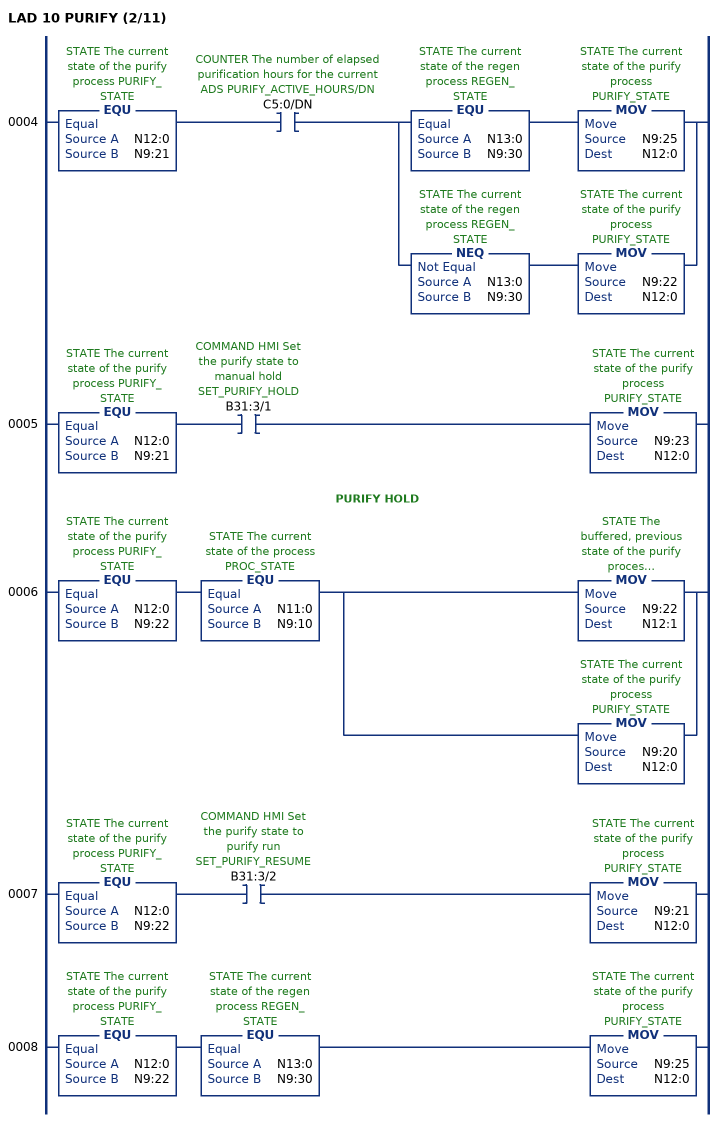
% Rung: 4 %
SOR EQU N12:0 N9:21 XIC C5:0/DN BST EQU N13:0 N9:30 MOV N9:25 N12:0 NXB NEQ N13:0 N9:30 MOV N9:22 N12:0 BND EOR
%   N12:0  PURIFY_STATE  "STATE The current state of the purify process" %
%   N9:21  PURIFY_RUN  "STATE Purify running" %
%   C5:0  PURIFY_ACTIVE_HOURS  "COUNTER The number of elapsed purification hours for the current ADS" %
%   N13:0  REGEN_STATE  "STATE The current state of the regen process" %
%   N9:30  REGEN_STANDBY  "STATE Regen Standby" %
%   N9:25  PURIFY_DONE %
%   N9:22  PURIFY_HOLD  "STATE Purify Hold" %
% Rung: 5 %
SOR EQU N12:0 N9:21 XIC B31:3/1 MOV N9:23 N12:0 EOR
%   N12:0  PURIFY_STATE  "STATE The current state of the purify process" %
%   N9:21  PURIFY_RUN  "STATE Purify running" %
%   B31:3/1  SET_PURIFY_HOLD  "COMMAND HMI Set the purify state to manual hold" %
%   N9:23  PURIFY_MANUAL_HOLD  "STATE Purify Manual Hold" %
% Rung: 6 %
% TITLE: PURIFY HOLD %
SOR EQU N12:0 N9:22 EQU N11:0 N9:10 BST MOV N9:22 N12:1 NXB MOV N9:20 N12:0 BND EOR
%   N12:0  PURIFY_STATE  "STATE The current state of the purify process" %
%   N9:22  PURIFY_HOLD  "STATE Purify Hold" %
%   N11:0  PROC_STATE  "STATE The current state of the process" %
%   N9:10  PROC_STANDBY  "STATE Process Standby" %
%   N12:1  PURIFY_STATE_BUFFER  "STATE The buffered, previous state of the purify process" %
%   N9:20  PURIFY_STANDBY  "STATE Purify Standby" %
% Rung: 7 %
SOR EQU N12:0 N9:22 XIC B31:3/2 MOV N9:21 N12:0 EOR
%   N12:0  PURIFY_STATE  "STATE The current state of the purify process" %
%   N9:22  PURIFY_HOLD  "STATE Purify Hold" %
%   B31:3/2  SET_PURIFY_RESUME  "COMMAND HMI Set the purify state to purify run" %
%   N9:21  PURIFY_RUN  "STATE Purify running" %
% Rung: 8 %
SOR EQU N12:0 N9:22 EQU N13:0 N9:30 MOV N9:25 N12:0 EOR
%   N12:0  PURIFY_STATE  "STATE The current state of the purify process" %
%   N9:22  PURIFY_HOLD  "STATE Purify Hold" %
%   N13:0  REGEN_STATE  "STATE The current state of the regen process" %
%   N9:30  REGEN_STANDBY  "STATE Regen Standby" %
%   N9:25  PURIFY_DONE %

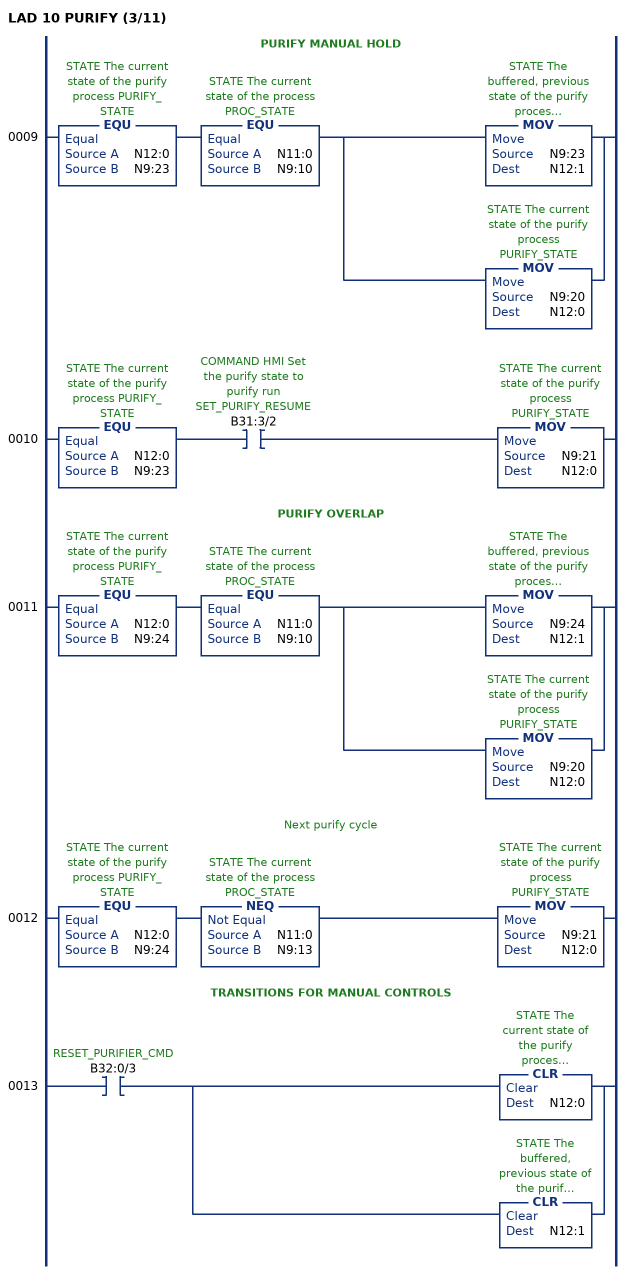
% Rung: 9 %
% TITLE: PURIFY MANUAL HOLD %
SOR EQU N12:0 N9:23 EQU N11:0 N9:10 BST MOV N9:23 N12:1 NXB MOV N9:20 N12:0 BND EOR
%   N12:0  PURIFY_STATE  "STATE The current state of the purify process" %
%   N9:23  PURIFY_MANUAL_HOLD  "STATE Purify Manual Hold" %
%   N11:0  PROC_STATE  "STATE The current state of the process" %
%   N9:10  PROC_STANDBY  "STATE Process Standby" %
%   N12:1  PURIFY_STATE_BUFFER  "STATE The buffered, previous state of the purify process" %
%   N9:20  PURIFY_STANDBY  "STATE Purify Standby" %
% Rung: 10 %
SOR EQU N12:0 N9:23 XIC B31:3/2 MOV N9:21 N12:0 EOR
%   N12:0  PURIFY_STATE  "STATE The current state of the purify process" %
%   N9:23  PURIFY_MANUAL_HOLD  "STATE Purify Manual Hold" %
%   B31:3/2  SET_PURIFY_RESUME  "COMMAND HMI Set the purify state to purify run" %
%   N9:21  PURIFY_RUN  "STATE Purify running" %
% Rung: 11 %
% TITLE: PURIFY OVERLAP %
SOR EQU N12:0 N9:24 EQU N11:0 N9:10 BST MOV N9:24 N12:1 NXB MOV N9:20 N12:0 BND EOR
%   N12:0  PURIFY_STATE  "STATE The current state of the purify process" %
%   N9:24  PURIFY_OVERLAP  "STATE Puriify Overlap" %
%   N11:0  PROC_STATE  "STATE The current state of the process" %
%   N9:10  PROC_STANDBY  "STATE Process Standby" %
%   N12:1  PURIFY_STATE_BUFFER  "STATE The buffered, previous state of the purify process" %
%   N9:20  PURIFY_STANDBY  "STATE Purify Standby" %
% Rung: 12 %
% Next purify cycle %
SOR EQU N12:0 N9:24 NEQ N11:0 N9:13 MOV N9:21 N12:0 EOR
%   N12:0  PURIFY_STATE  "STATE The current state of the purify process" %
%   N9:24  PURIFY_OVERLAP  "STATE Puriify Overlap" %
%   N11:0  PROC_STATE  "STATE The current state of the process" %
%   N9:13  PROC_OVERLAP  "STATE Process Purify Overlap" %
%   N9:21  PURIFY_RUN  "STATE Purify running" %
% Rung: 13 %
% TITLE: TRANSITIONS FOR MANUAL CONTROLS %
SOR XIC B32:0/3 BST CLR N12:0 NXB CLR N12:1 BND EOR
%   B32:0/3  RESET_PURIFIER_CMD %
%   N12:0  PURIFY_STATE  "STATE The current state of the purify process" %
%   N12:1  PURIFY_STATE_BUFFER  "STATE The buffered, previous state of the purify process" %

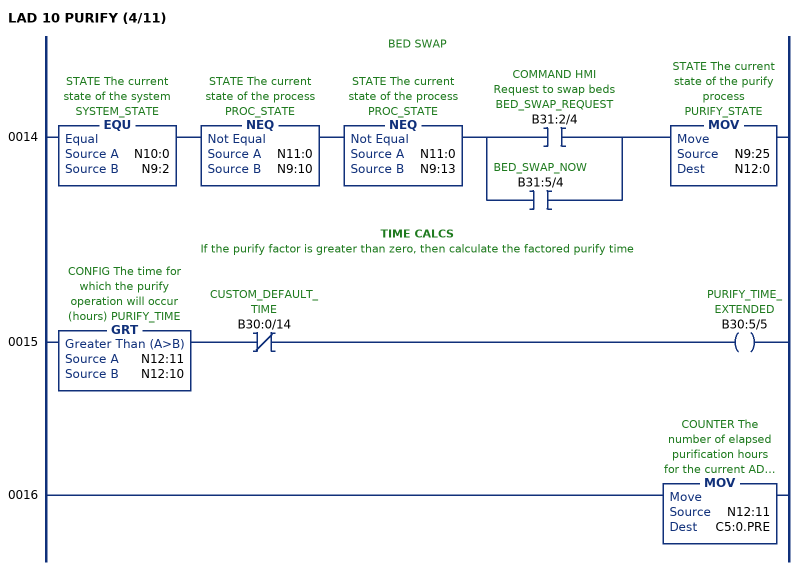
% Rung: 14 %
% BED SWAP %
SOR EQU N10:0 N9:2 NEQ N11:0 N9:10 NEQ N11:0 N9:13 BST XIC B31:2/4 NXB XIC B31:5/4 BND MOV N9:25 N12:0 EOR
%   N10:0  SYSTEM_STATE  "STATE The current state of the system" %
%   N9:2  SYSTEM_PROCESS  "STATE System Process" %
%   N11:0  PROC_STATE  "STATE The current state of the process" %
%   N9:10  PROC_STANDBY  "STATE Process Standby" %
%   N9:13  PROC_OVERLAP  "STATE Process Purify Overlap" %
%   B31:2/4  BED_SWAP_REQUEST  "COMMAND HMI Request to swap beds" %
%   B31:5/4  BED_SWAP_NOW %
%   N9:25  PURIFY_DONE %
%   N12:0  PURIFY_STATE  "STATE The current state of the purify process" %
% Rung: 15 %
% TITLE: TIME CALCS %
% If the purify factor is greater than zero, then calculate the factored purify time %
SOR GRT N12:11 N12:10 XIO B30:0/14 OTE B30:5/5 EOR
%   N12:11  PURIFY_TIME  "CONFIG The time for which the purify operation will occur (hours)" %
%   N12:10  DEFAULT_PURIFY_TIME %
%   B30:0/14  CUSTOM_DEFAULT_TIME %
%   B30:5/5  PURIFY_TIME_EXTENDED %
% Rung: 16 %
SOR MOV N12:11 C5:0.PRE EOR
%   N12:11  PURIFY_TIME  "CONFIG The time for which the purify operation will occur (hours)" %
%   C5:0  PURIFY_ACTIVE_HOURS  "COUNTER The number of elapsed purification hours for the current ADS" %

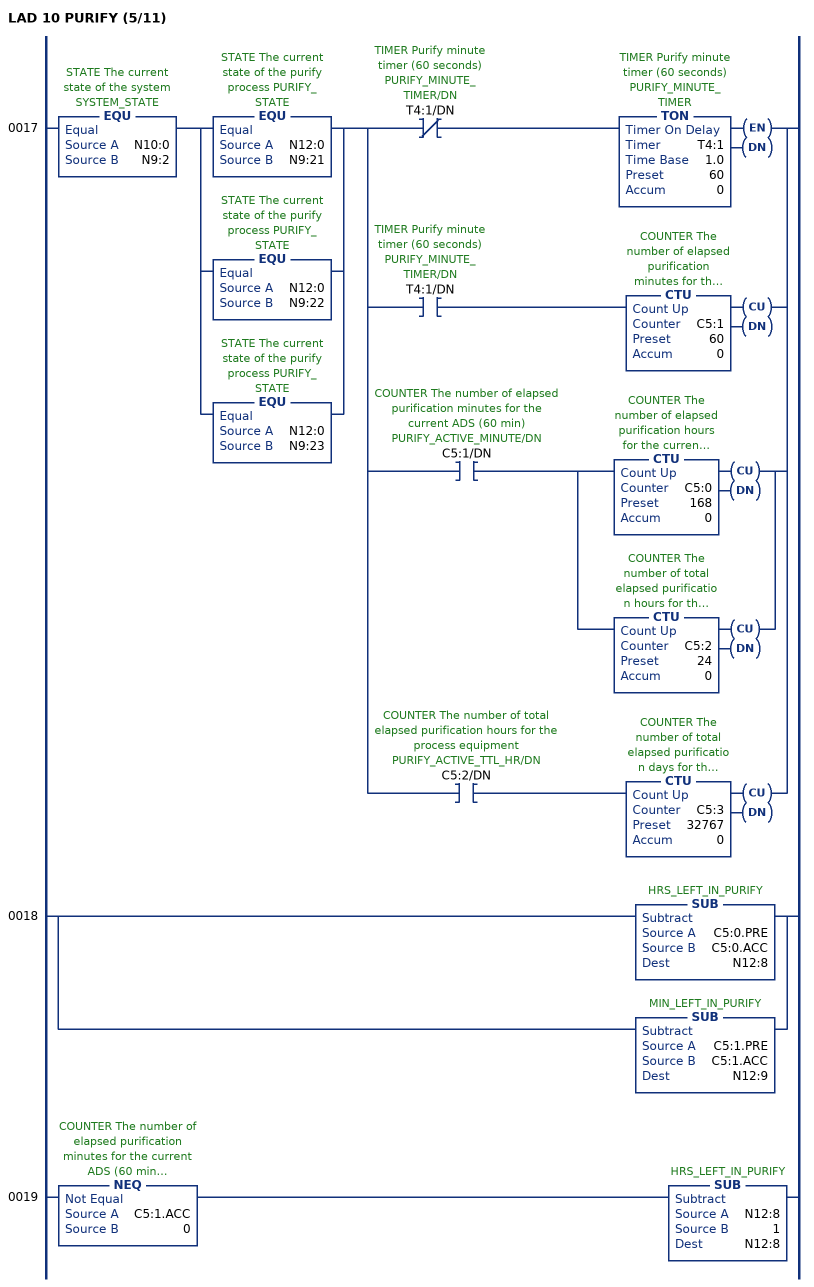
% Rung: 17 %
SOR EQU N10:0 N9:2 BST EQU N12:0 N9:21 NXB EQU N12:0 N9:22 NXB EQU N12:0 N9:23 BND BST XIO T4:1/DN TON T4:1 1.0 60 0 NXB XIC T4:1/DN CTU C5:1 60 0 NXB XIC C5:1/DN BST CTU C5:0 168 0 NXB CTU C5:2 24 0 BND NXB XIC C5:2/DN CTU C5:3 32767 0 BND EOR
%   N10:0  SYSTEM_STATE  "STATE The current state of the system" %
%   N9:2  SYSTEM_PROCESS  "STATE System Process" %
%   N12:0  PURIFY_STATE  "STATE The current state of the purify process" %
%   N9:21  PURIFY_RUN  "STATE Purify running" %
%   N9:22  PURIFY_HOLD  "STATE Purify Hold" %
%   N9:23  PURIFY_MANUAL_HOLD  "STATE Purify Manual Hold" %
%   T4:1  PURIFY_MINUTE_TIMER  "TIMER Purify minute timer (60 seconds)" %
%   C5:1  PURIFY_ACTIVE_MINUTE  "COUNTER The number of elapsed purification minutes for the current ADS (60 min)" %
%   C5:0  PURIFY_ACTIVE_HOURS  "COUNTER The number of elapsed purification hours for the current ADS" %
%   C5:2  PURIFY_ACTIVE_TTL_HR  "COUNTER The number of total elapsed purification hours for the process equipment" %
%   C5:3  PURIFY_ACTIVE_TTL_DY  "COUNTER The number of total elapsed purification days for the process equipment" %
% Rung: 18 %
SOR BST SUB C5:0.PRE C5:0.ACC N12:8 NXB SUB C5:1.PRE C5:1.ACC N12:9 BND EOR
%   C5:0  PURIFY_ACTIVE_HOURS  "COUNTER The number of elapsed purification hours for the current ADS" %
%   N12:8  HRS_LEFT_IN_PURIFY %
%   C5:1  PURIFY_ACTIVE_MINUTE  "COUNTER The number of elapsed purification minutes for the current ADS (60 min)" %
%   N12:9  MIN_LEFT_IN_PURIFY %
% Rung: 19 %
SOR NEQ C5:1.ACC 0 SUB N12:8 1 N12:8 EOR
%   C5:1  PURIFY_ACTIVE_MINUTE  "COUNTER The number of elapsed purification minutes for the current ADS (60 min)" %
%   N12:8  HRS_LEFT_IN_PURIFY %

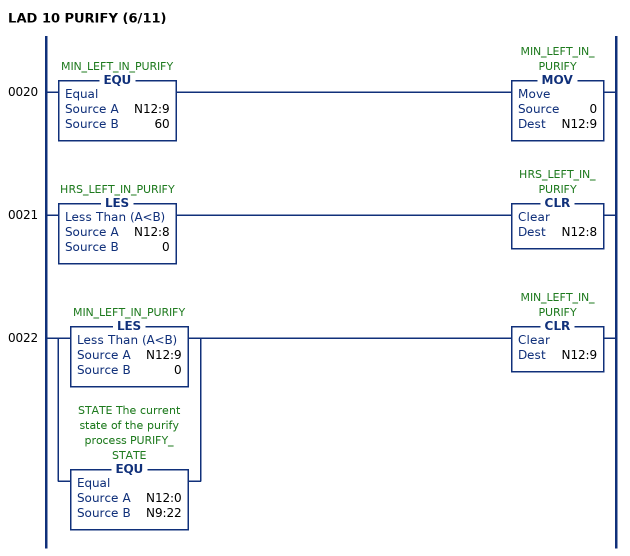
% Rung: 20 %
SOR EQU N12:9 60 MOV 0 N12:9 EOR
%   N12:9  MIN_LEFT_IN_PURIFY %
% Rung: 21 %
SOR LES N12:8 0 CLR N12:8 EOR
%   N12:8  HRS_LEFT_IN_PURIFY %
% Rung: 22 %
SOR BST LES N12:9 0 NXB EQU N12:0 N9:22 BND CLR N12:9 EOR
%   N12:9  MIN_LEFT_IN_PURIFY %
%   N12:0  PURIFY_STATE  "STATE The current state of the purify process" %
%   N9:22  PURIFY_HOLD  "STATE Purify Hold" %

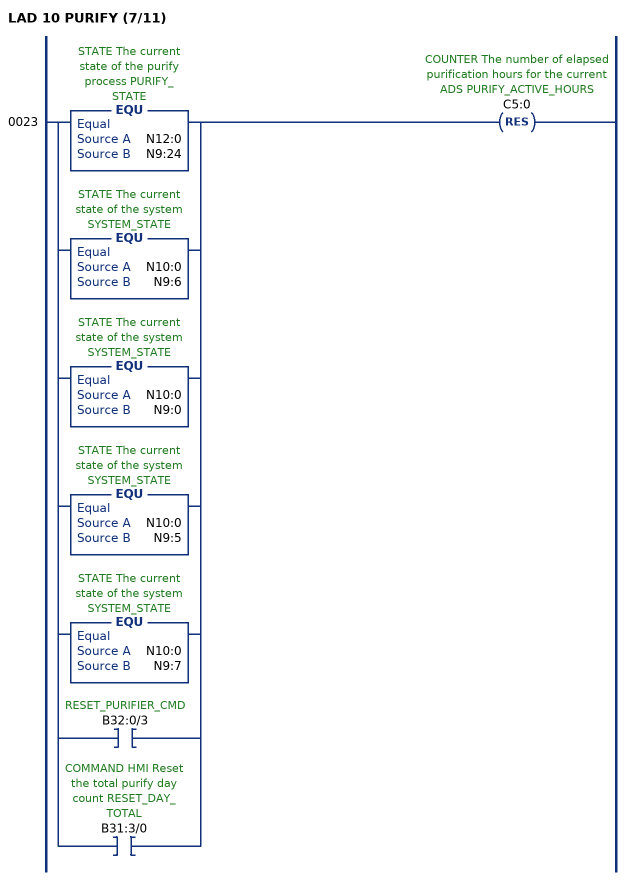
% Rung: 23 %
SOR BST EQU N12:0 N9:24 NXB EQU N10:0 N9:6 NXB EQU N10:0 N9:0 NXB EQU N10:0 N9:5 NXB EQU N10:0 N9:7 NXB XIC B32:0/3 NXB XIC B31:3/0 BND RES C5:0 EOR
%   N12:0  PURIFY_STATE  "STATE The current state of the purify process" %
%   N9:24  PURIFY_OVERLAP  "STATE Puriify Overlap" %
%   N10:0  SYSTEM_STATE  "STATE The current state of the system" %
%   N9:6  SYSTEM_PURGE %
%   N9:0  SYSTEM_OFFLINE %
%   N9:5  SYSTEM_QUICK_START %
%   N9:7  SYSTEM_COLD_START %
%   B32:0/3  RESET_PURIFIER_CMD %
%   B31:3/0  RESET_DAY_TOTAL  "COMMAND HMI Reset the total purify day count" %
%   C5:0  PURIFY_ACTIVE_HOURS  "COUNTER The number of elapsed purification hours for the current ADS" %

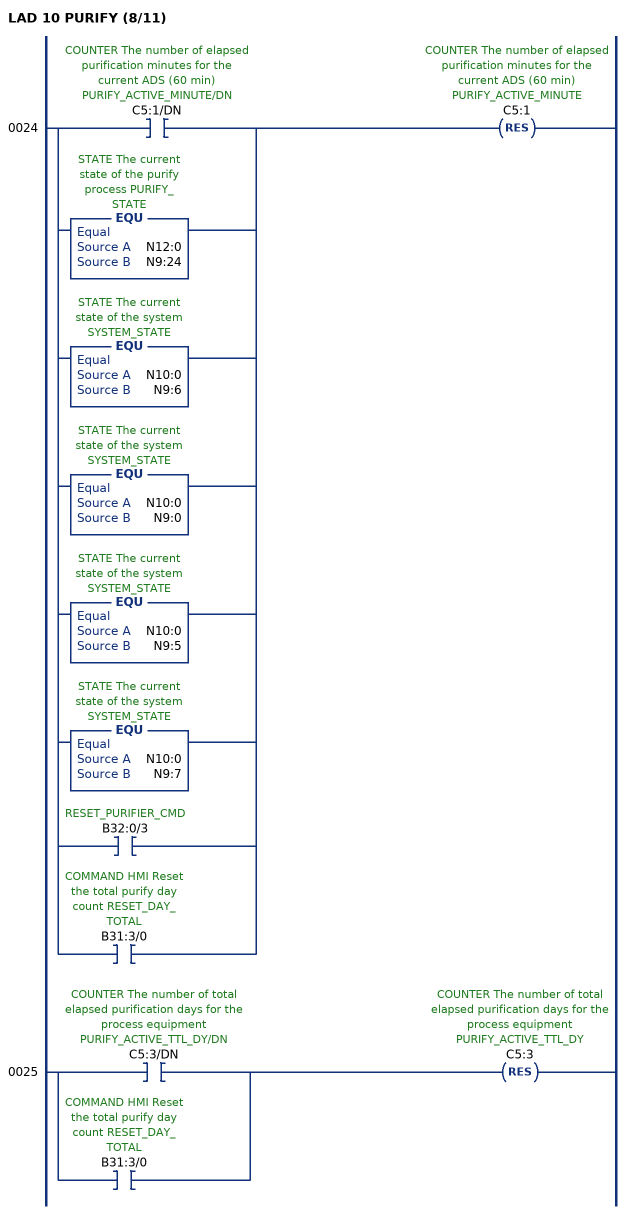
% Rung: 24 %
SOR BST XIC C5:1/DN NXB EQU N12:0 N9:24 NXB EQU N10:0 N9:6 NXB EQU N10:0 N9:0 NXB EQU N10:0 N9:5 NXB EQU N10:0 N9:7 NXB XIC B32:0/3 NXB XIC B31:3/0 BND RES C5:1 EOR
%   C5:1  PURIFY_ACTIVE_MINUTE  "COUNTER The number of elapsed purification minutes for the current ADS (60 min)" %
%   N12:0  PURIFY_STATE  "STATE The current state of the purify process" %
%   N9:24  PURIFY_OVERLAP  "STATE Puriify Overlap" %
%   N10:0  SYSTEM_STATE  "STATE The current state of the system" %
%   N9:6  SYSTEM_PURGE %
%   N9:0  SYSTEM_OFFLINE %
%   N9:5  SYSTEM_QUICK_START %
%   N9:7  SYSTEM_COLD_START %
%   B32:0/3  RESET_PURIFIER_CMD %
%   B31:3/0  RESET_DAY_TOTAL  "COMMAND HMI Reset the total purify day count" %
% Rung: 25 %
SOR BST XIC C5:3/DN NXB XIC B31:3/0 BND RES C5:3 EOR
%   C5:3  PURIFY_ACTIVE_TTL_DY  "COUNTER The number of total elapsed purification days for the process equipment" %
%   B31:3/0  RESET_DAY_TOTAL  "COMMAND HMI Reset the total purify day count" %

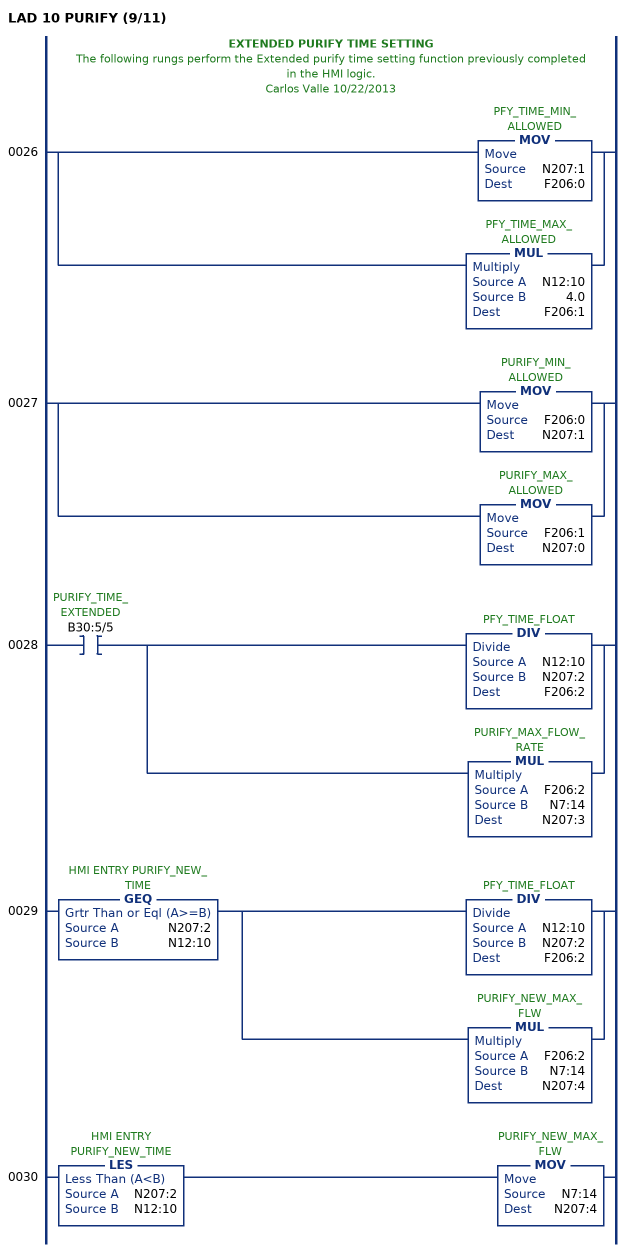
% Rung: 26 %
% TITLE: EXTENDED PURIFY TIME SETTING %
% The following rungs perform the Extended purify time setting function previously completed in the HMI logic.
% Carlos Valle 10/22/2013 %
SOR BST MOV N207:1 F206:0 NXB MUL N12:10 4.0 F206:1 BND EOR
%   N207:1  PURIFY_MIN_ALLOWED %
%   F206:0  PFY_TIME_MIN_ALLOWED %
%   N12:10  DEFAULT_PURIFY_TIME %
%   F206:1  PFY_TIME_MAX_ALLOWED %
% Rung: 27 %
SOR BST MOV F206:0 N207:1 NXB MOV F206:1 N207:0 BND EOR
%   F206:0  PFY_TIME_MIN_ALLOWED %
%   N207:1  PURIFY_MIN_ALLOWED %
%   F206:1  PFY_TIME_MAX_ALLOWED %
%   N207:0  PURIFY_MAX_ALLOWED %
% Rung: 28 %
SOR XIC B30:5/5 BST DIV N12:10 N207:2 F206:2 NXB MUL F206:2 N7:14 N207:3 BND EOR
%   B30:5/5  PURIFY_TIME_EXTENDED %
%   N12:10  DEFAULT_PURIFY_TIME %
%   N207:2  PURIFY_NEW_TIME  "HMI ENTRY" %
%   F206:2  PFY_TIME_FLOAT %
%   N7:14  PURIFIER_SIZE %
%   N207:3  PURIFY_MAX_FLOW_RATE %
% Rung: 29 %
SOR GEQ N207:2 N12:10 BST DIV N12:10 N207:2 F206:2 NXB MUL F206:2 N7:14 N207:4 BND EOR
%   N207:2  PURIFY_NEW_TIME  "HMI ENTRY" %
%   N12:10  DEFAULT_PURIFY_TIME %
%   F206:2  PFY_TIME_FLOAT %
%   N7:14  PURIFIER_SIZE %
%   N207:4  PURIFY_NEW_MAX_FLW %
% Rung: 30 %
SOR LES N207:2 N12:10 MOV N7:14 N207:4 EOR
%   N207:2  PURIFY_NEW_TIME  "HMI ENTRY" %
%   N12:10  DEFAULT_PURIFY_TIME %
%   N7:14  PURIFIER_SIZE %
%   N207:4  PURIFY_NEW_MAX_FLW %

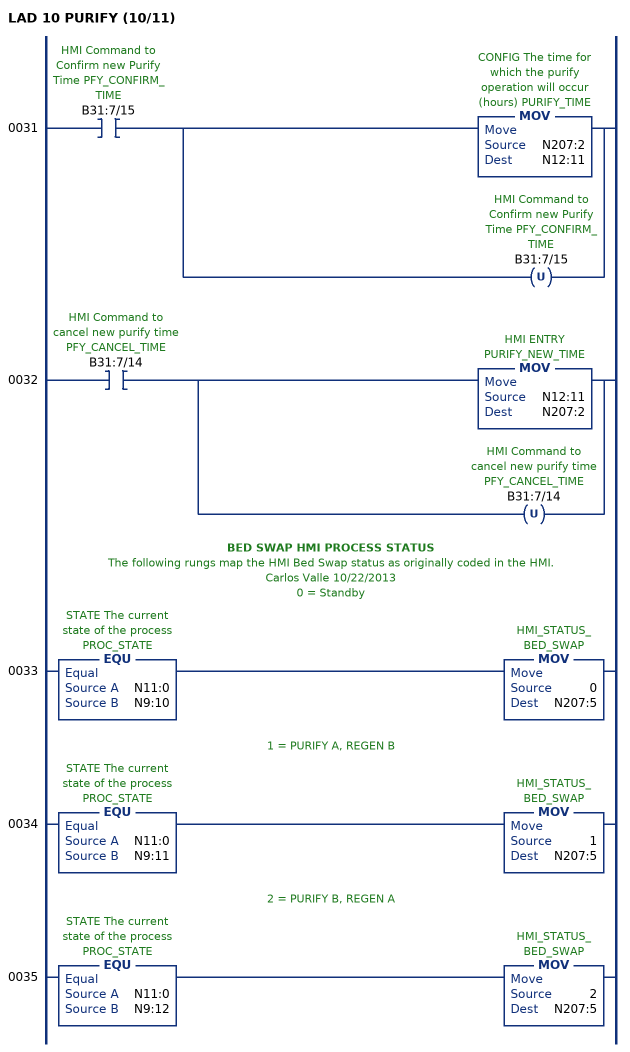
% Rung: 31 %
SOR XIC B31:7/15 BST MOV N207:2 N12:11 NXB OTU B31:7/15 BND EOR
%   B31:7/15  PFY_CONFIRM_TIME  "HMI Command to Confirm new Purify Time" %
%   N207:2  PURIFY_NEW_TIME  "HMI ENTRY" %
%   N12:11  PURIFY_TIME  "CONFIG The time for which the purify operation will occur (hours)" %
% Rung: 32 %
SOR XIC B31:7/14 BST MOV N12:11 N207:2 NXB OTU B31:7/14 BND EOR
%   B31:7/14  PFY_CANCEL_TIME  "HMI Command to cancel new purify time" %
%   N12:11  PURIFY_TIME  "CONFIG The time for which the purify operation will occur (hours)" %
%   N207:2  PURIFY_NEW_TIME  "HMI ENTRY" %
% Rung: 33 %
% TITLE: BED SWAP HMI PROCESS STATUS %
% The following rungs map the HMI Bed Swap status as originally coded in the HMI.
% Carlos Valle 10/22/2013
% 0 = Standby %
SOR EQU N11:0 N9:10 MOV 0 N207:5 EOR
%   N11:0  PROC_STATE  "STATE The current state of the process" %
%   N9:10  PROC_STANDBY  "STATE Process Standby" %
%   N207:5  HMI_STATUS_BED_SWAP %
% Rung: 34 %
% 1 = PURIFY A, REGEN B %
SOR EQU N11:0 N9:11 MOV 1 N207:5 EOR
%   N11:0  PROC_STATE  "STATE The current state of the process" %
%   N9:11  PROC_PFY_A_REG_B  "STATE Process Purify A" %
%   N207:5  HMI_STATUS_BED_SWAP %
% Rung: 35 %
% 2 = PURIFY B, REGEN A %
SOR EQU N11:0 N9:12 MOV 2 N207:5 EOR
%   N11:0  PROC_STATE  "STATE The current state of the process" %
%   N9:12  PROC_PFY_B_REG_A  "STATE Process Purify B" %
%   N207:5  HMI_STATUS_BED_SWAP %

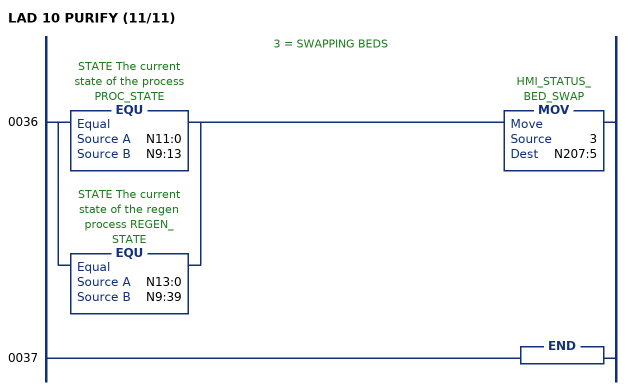
% Rung: 36 %
% 3 = SWAPPING BEDS %
SOR BST EQU N11:0 N9:13 NXB EQU N13:0 N9:39 BND MOV 3 N207:5 EOR
%   N11:0  PROC_STATE  "STATE The current state of the process" %
%   N9:13  PROC_OVERLAP  "STATE Process Purify Overlap" %
%   N13:0  REGEN_STATE  "STATE The current state of the regen process" %
%   N9:39  REGEN_BACKFILL %
%   N207:5  HMI_STATUS_BED_SWAP %
% Rung: 37 %
SOR END EOR

LADDER 11 "REGEN"    % Operates the regen control %
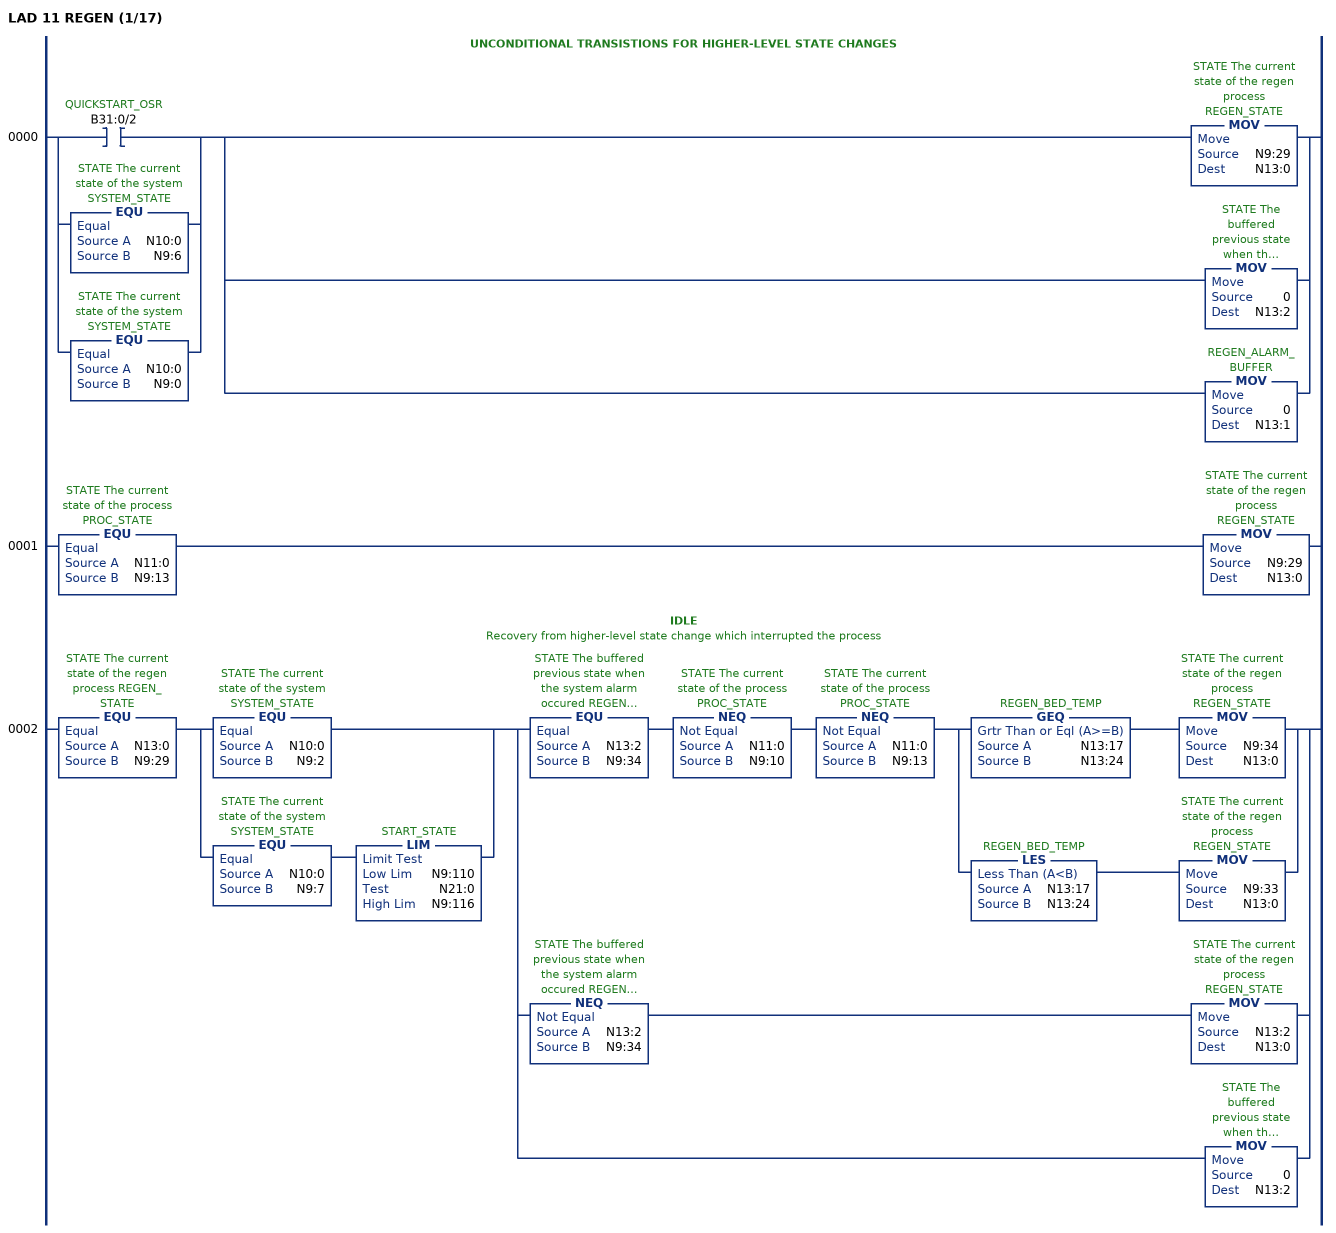
% Rung: 0 %
% TITLE: UNCONDITIONAL TRANSISTIONS FOR HIGHER-LEVEL STATE CHANGES %
SOR BST XIC B31:0/2 NXB EQU N10:0 N9:6 NXB EQU N10:0 N9:0 BND BST MOV N9:29 N13:0 NXB MOV 0 N13:2 NXB MOV 0 N13:1 BND EOR
%   B31:0/2  QUICKSTART_OSR %
%   N10:0  SYSTEM_STATE  "STATE The current state of the system" %
%   N9:6  SYSTEM_PURGE %
%   N9:0  SYSTEM_OFFLINE %
%   N9:29  REGEN_IDLE %
%   N13:0  REGEN_STATE  "STATE The current state of the regen process" %
%   N13:2  REGEN_SYSTEM_BUFFER  "STATE The buffered previous state when the system alarm occured" %
%   N13:1  REGEN_ALARM_BUFFER %
% Rung: 1 %
SOR EQU N11:0 N9:13 MOV N9:29 N13:0 EOR
%   N11:0  PROC_STATE  "STATE The current state of the process" %
%   N9:13  PROC_OVERLAP  "STATE Process Purify Overlap" %
%   N9:29  REGEN_IDLE %
%   N13:0  REGEN_STATE  "STATE The current state of the regen process" %
% Rung: 2 %
% TITLE: IDLE %
% Recovery from higher-level state change which interrupted the process %
SOR EQU N13:0 N9:29 BST EQU N10:0 N9:2 NXB EQU N10:0 N9:7 LIM N9:110 N21:0 N9:116 BND BST EQU N13:2 N9:34 NEQ N11:0 N9:10 NEQ N11:0 N9:13 BST GEQ N13:17 N13:24 MOV N9:34 N13:0 NXB LES N13:17 N13:24 MOV N9:33 N13:0 BND NXB NEQ N13:2 N9:34 MOV N13:2 N13:0 NXB MOV 0 N13:2 BND EOR
%   N13:0  REGEN_STATE  "STATE The current state of the regen process" %
%   N9:29  REGEN_IDLE %
%   N10:0  SYSTEM_STATE  "STATE The current state of the system" %
%   N9:2  SYSTEM_PROCESS  "STATE System Process" %
%   N9:7  SYSTEM_COLD_START %
%   N9:110  START_REG_VENT %
%   N21:0  START_STATE %
%   N9:116  START_REG_BACKFILL %
%   N13:2  REGEN_SYSTEM_BUFFER  "STATE The buffered previous state when the system alarm occured" %
%   N9:34  REGEN_RUN  "STATE Regen Running" %
%   N11:0  PROC_STATE  "STATE The current state of the process" %
%   N9:10  PROC_STANDBY  "STATE Process Standby" %
%   N9:13  PROC_OVERLAP  "STATE Process Purify Overlap" %
%   N13:17  REGEN_BED_TEMP %
%   N13:24  ADS_BED_TEMP_HIGH  "CONFIG The temp at which the regen process may continue" %
%   N9:33  REGEN_HEAT_BED  "STATE Regen Heat wall" %

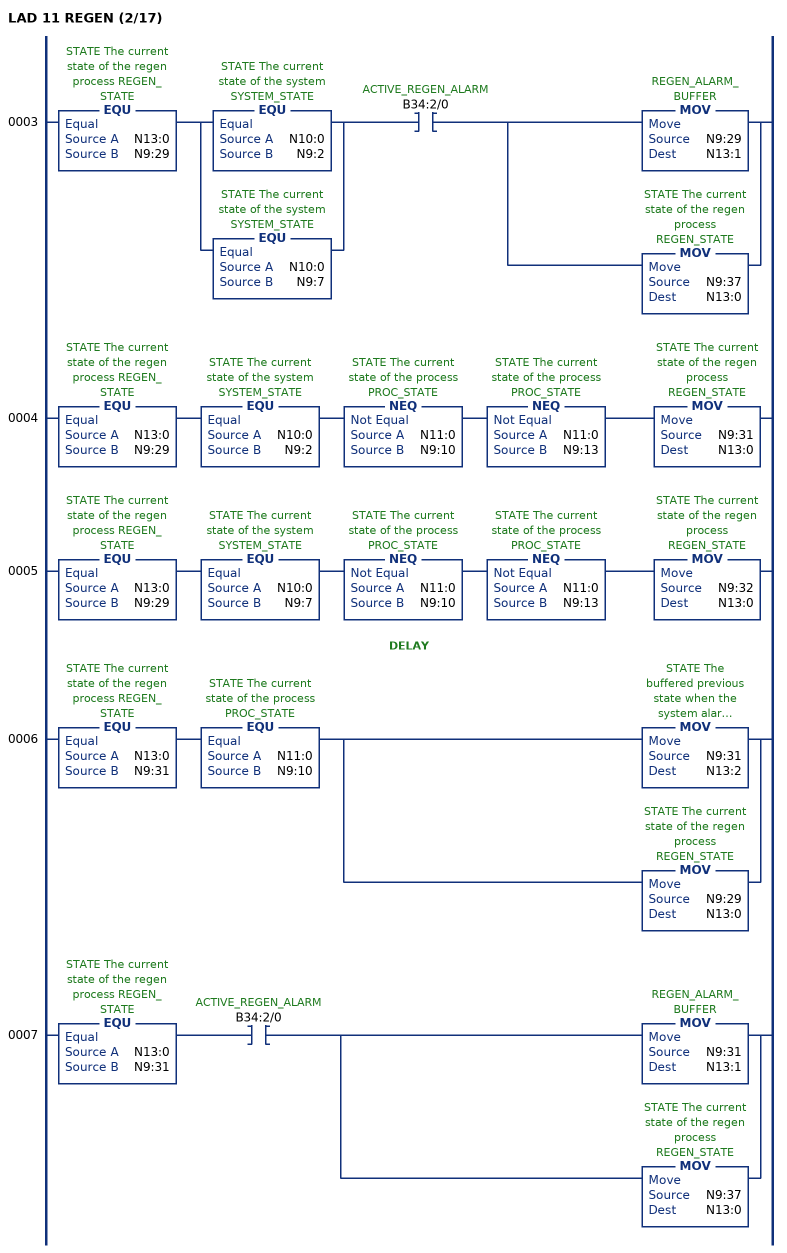
% Rung: 3 %
SOR EQU N13:0 N9:29 BST EQU N10:0 N9:2 NXB EQU N10:0 N9:7 BND XIC B34:2/0 BST MOV N9:29 N13:1 NXB MOV N9:37 N13:0 BND EOR
%   N13:0  REGEN_STATE  "STATE The current state of the regen process" %
%   N9:29  REGEN_IDLE %
%   N10:0  SYSTEM_STATE  "STATE The current state of the system" %
%   N9:2  SYSTEM_PROCESS  "STATE System Process" %
%   N9:7  SYSTEM_COLD_START %
%   B34:2/0  ACTIVE_REGEN_ALARM %
%   N13:1  REGEN_ALARM_BUFFER %
%   N9:37  REGEN_ALARM  "STATE Regen Alarm" %
% Rung: 4 %
SOR EQU N13:0 N9:29 EQU N10:0 N9:2 NEQ N11:0 N9:10 NEQ N11:0 N9:13 MOV N9:31 N13:0 EOR
%   N13:0  REGEN_STATE  "STATE The current state of the regen process" %
%   N9:29  REGEN_IDLE %
%   N10:0  SYSTEM_STATE  "STATE The current state of the system" %
%   N9:2  SYSTEM_PROCESS  "STATE System Process" %
%   N11:0  PROC_STATE  "STATE The current state of the process" %
%   N9:10  PROC_STANDBY  "STATE Process Standby" %
%   N9:13  PROC_OVERLAP  "STATE Process Purify Overlap" %
%   N9:31  REGEN_DELAY  "STATE Regen Delay" %
% Rung: 5 %
SOR EQU N13:0 N9:29 EQU N10:0 N9:7 NEQ N11:0 N9:10 NEQ N11:0 N9:13 MOV N9:32 N13:0 EOR
%   N13:0  REGEN_STATE  "STATE The current state of the regen process" %
%   N9:29  REGEN_IDLE %
%   N10:0  SYSTEM_STATE  "STATE The current state of the system" %
%   N9:7  SYSTEM_COLD_START %
%   N11:0  PROC_STATE  "STATE The current state of the process" %
%   N9:10  PROC_STANDBY  "STATE Process Standby" %
%   N9:13  PROC_OVERLAP  "STATE Process Purify Overlap" %
%   N9:32  REGEN_VENT  "STATE Regen Vent" %
% Rung: 6 %
% TITLE: DELAY %
SOR EQU N13:0 N9:31 EQU N11:0 N9:10 BST MOV N9:31 N13:2 NXB MOV N9:29 N13:0 BND EOR
%   N13:0  REGEN_STATE  "STATE The current state of the regen process" %
%   N9:31  REGEN_DELAY  "STATE Regen Delay" %
%   N11:0  PROC_STATE  "STATE The current state of the process" %
%   N9:10  PROC_STANDBY  "STATE Process Standby" %
%   N13:2  REGEN_SYSTEM_BUFFER  "STATE The buffered previous state when the system alarm occured" %
%   N9:29  REGEN_IDLE %
% Rung: 7 %
SOR EQU N13:0 N9:31 XIC B34:2/0 BST MOV N9:31 N13:1 NXB MOV N9:37 N13:0 BND EOR
%   N13:0  REGEN_STATE  "STATE The current state of the regen process" %
%   N9:31  REGEN_DELAY  "STATE Regen Delay" %
%   B34:2/0  ACTIVE_REGEN_ALARM %
%   N13:1  REGEN_ALARM_BUFFER %
%   N9:37  REGEN_ALARM  "STATE Regen Alarm" %

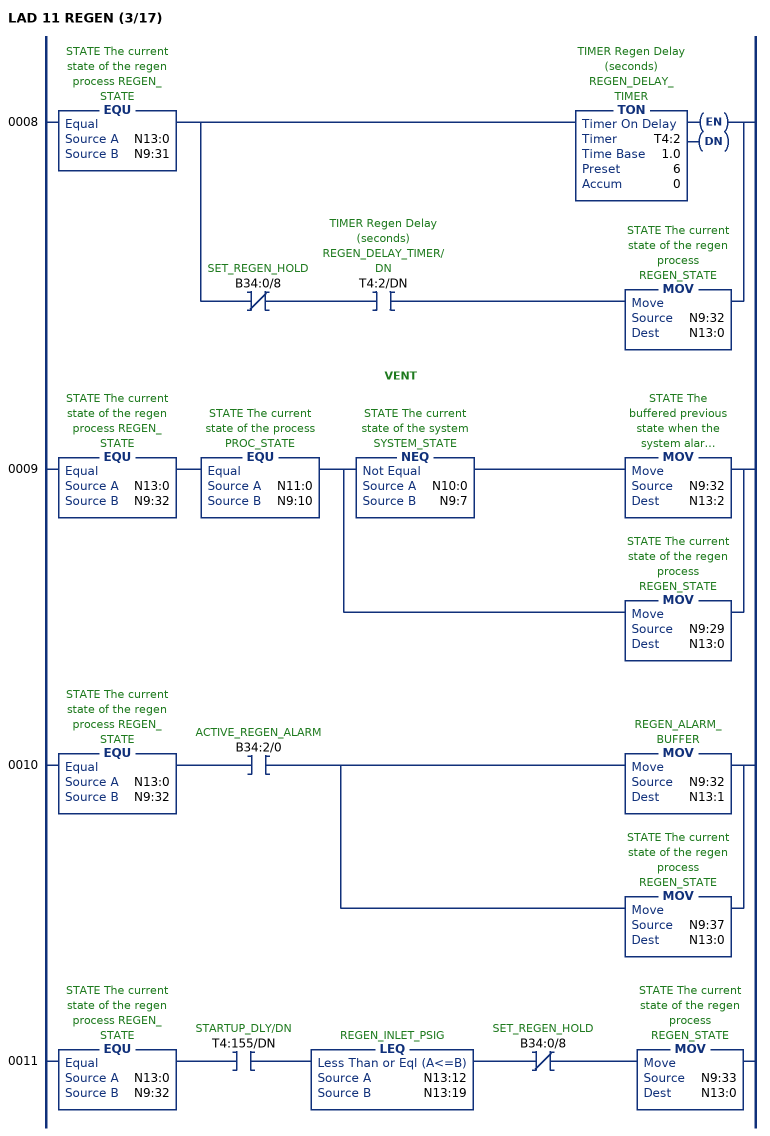
% Rung: 8 %
SOR EQU N13:0 N9:31 BST TON T4:2 1.0 6 0 NXB XIO B34:0/8 XIC T4:2/DN MOV N9:32 N13:0 BND EOR
%   N13:0  REGEN_STATE  "STATE The current state of the regen process" %
%   N9:31  REGEN_DELAY  "STATE Regen Delay" %
%   T4:2  REGEN_DELAY_TIMER  "TIMER Regen Delay (seconds)" %
%   B34:0/8  SET_REGEN_HOLD %
%   N9:32  REGEN_VENT  "STATE Regen Vent" %
% Rung: 9 %
% TITLE: VENT %
SOR EQU N13:0 N9:32 EQU N11:0 N9:10 BST NEQ N10:0 N9:7 MOV N9:32 N13:2 NXB MOV N9:29 N13:0 BND EOR
%   N13:0  REGEN_STATE  "STATE The current state of the regen process" %
%   N9:32  REGEN_VENT  "STATE Regen Vent" %
%   N11:0  PROC_STATE  "STATE The current state of the process" %
%   N9:10  PROC_STANDBY  "STATE Process Standby" %
%   N10:0  SYSTEM_STATE  "STATE The current state of the system" %
%   N9:7  SYSTEM_COLD_START %
%   N13:2  REGEN_SYSTEM_BUFFER  "STATE The buffered previous state when the system alarm occured" %
%   N9:29  REGEN_IDLE %
% Rung: 10 %
SOR EQU N13:0 N9:32 XIC B34:2/0 BST MOV N9:32 N13:1 NXB MOV N9:37 N13:0 BND EOR
%   N13:0  REGEN_STATE  "STATE The current state of the regen process" %
%   N9:32  REGEN_VENT  "STATE Regen Vent" %
%   B34:2/0  ACTIVE_REGEN_ALARM %
%   N13:1  REGEN_ALARM_BUFFER %
%   N9:37  REGEN_ALARM  "STATE Regen Alarm" %
% Rung: 11 %
SOR EQU N13:0 N9:32 XIC T4:155/DN LEQ N13:12 N13:19 XIO B34:0/8 MOV N9:33 N13:0 EOR
%   N13:0  REGEN_STATE  "STATE The current state of the regen process" %
%   N9:32  REGEN_VENT  "STATE Regen Vent" %
%   T4:155  STARTUP_DLY %
%   N13:12  REGEN_INLET_PSIG %
%   N13:19  REGEN_VENT_PRES %
%   B34:0/8  SET_REGEN_HOLD %
%   N9:33  REGEN_HEAT_BED  "STATE Regen Heat wall" %

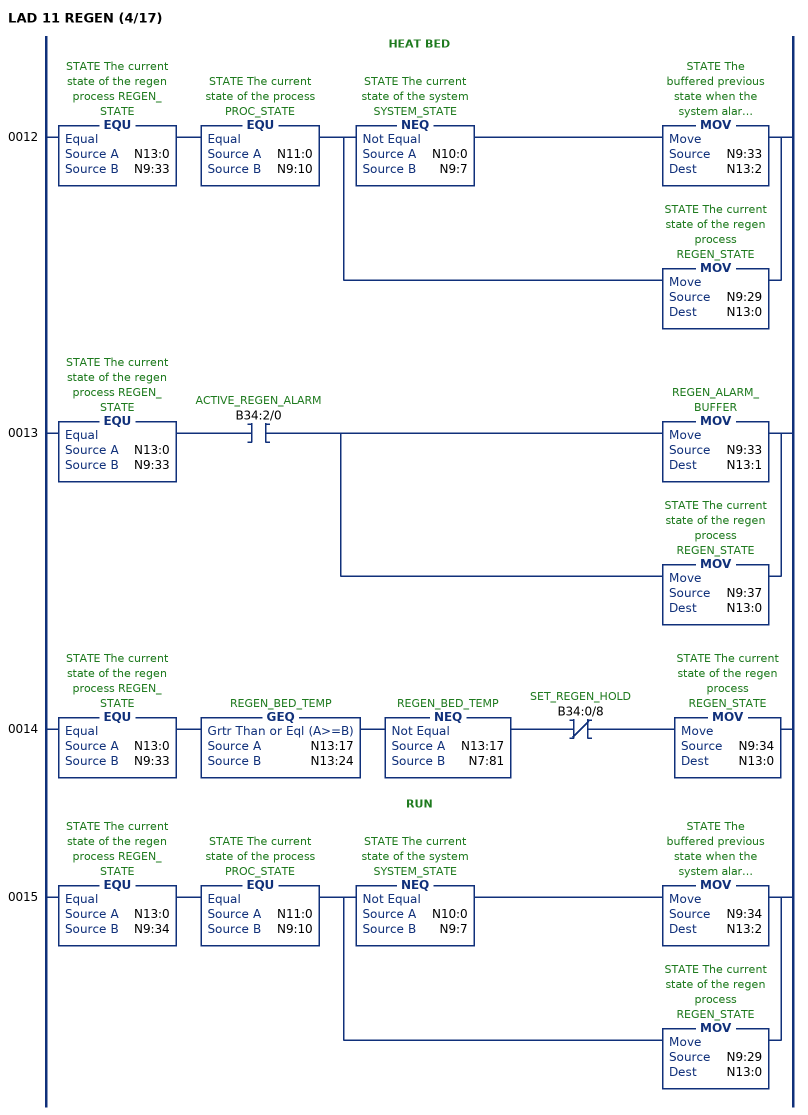
% Rung: 12 %
% TITLE: HEAT BED %
SOR EQU N13:0 N9:33 EQU N11:0 N9:10 BST NEQ N10:0 N9:7 MOV N9:33 N13:2 NXB MOV N9:29 N13:0 BND EOR
%   N13:0  REGEN_STATE  "STATE The current state of the regen process" %
%   N9:33  REGEN_HEAT_BED  "STATE Regen Heat wall" %
%   N11:0  PROC_STATE  "STATE The current state of the process" %
%   N9:10  PROC_STANDBY  "STATE Process Standby" %
%   N10:0  SYSTEM_STATE  "STATE The current state of the system" %
%   N9:7  SYSTEM_COLD_START %
%   N13:2  REGEN_SYSTEM_BUFFER  "STATE The buffered previous state when the system alarm occured" %
%   N9:29  REGEN_IDLE %
% Rung: 13 %
SOR EQU N13:0 N9:33 XIC B34:2/0 BST MOV N9:33 N13:1 NXB MOV N9:37 N13:0 BND EOR
%   N13:0  REGEN_STATE  "STATE The current state of the regen process" %
%   N9:33  REGEN_HEAT_BED  "STATE Regen Heat wall" %
%   B34:2/0  ACTIVE_REGEN_ALARM %
%   N13:1  REGEN_ALARM_BUFFER %
%   N9:37  REGEN_ALARM  "STATE Regen Alarm" %
% Rung: 14 %
SOR EQU N13:0 N9:33 GEQ N13:17 N13:24 NEQ N13:17 N7:81 XIO B34:0/8 MOV N9:34 N13:0 EOR
%   N13:0  REGEN_STATE  "STATE The current state of the regen process" %
%   N9:33  REGEN_HEAT_BED  "STATE Regen Heat wall" %
%   N13:17  REGEN_BED_TEMP %
%   N13:24  ADS_BED_TEMP_HIGH  "CONFIG The temp at which the regen process may continue" %
%   N7:81  TC_OPEN_SP  "CONFIG The value read by an open TC input" %
%   B34:0/8  SET_REGEN_HOLD %
%   N9:34  REGEN_RUN  "STATE Regen Running" %
% Rung: 15 %
% TITLE: RUN %
SOR EQU N13:0 N9:34 EQU N11:0 N9:10 BST NEQ N10:0 N9:7 MOV N9:34 N13:2 NXB MOV N9:29 N13:0 BND EOR
%   N13:0  REGEN_STATE  "STATE The current state of the regen process" %
%   N9:34  REGEN_RUN  "STATE Regen Running" %
%   N11:0  PROC_STATE  "STATE The current state of the process" %
%   N9:10  PROC_STANDBY  "STATE Process Standby" %
%   N10:0  SYSTEM_STATE  "STATE The current state of the system" %
%   N9:7  SYSTEM_COLD_START %
%   N13:2  REGEN_SYSTEM_BUFFER  "STATE The buffered previous state when the system alarm occured" %
%   N9:29  REGEN_IDLE %

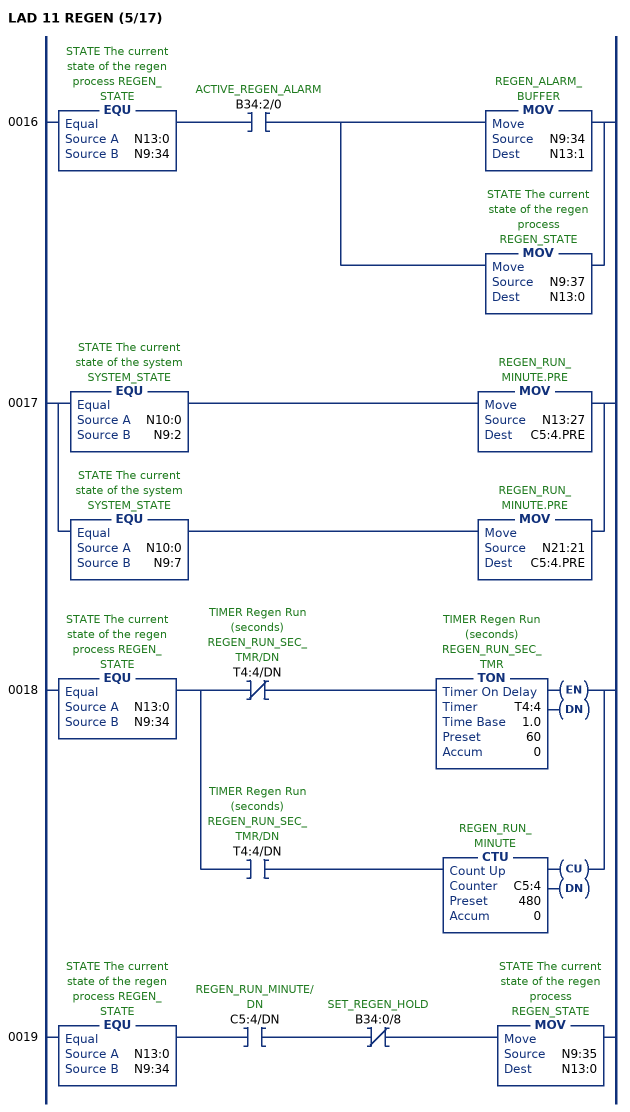
% Rung: 16 %
SOR EQU N13:0 N9:34 XIC B34:2/0 BST MOV N9:34 N13:1 NXB MOV N9:37 N13:0 BND EOR
%   N13:0  REGEN_STATE  "STATE The current state of the regen process" %
%   N9:34  REGEN_RUN  "STATE Regen Running" %
%   B34:2/0  ACTIVE_REGEN_ALARM %
%   N13:1  REGEN_ALARM_BUFFER %
%   N9:37  REGEN_ALARM  "STATE Regen Alarm" %
% Rung: 17 %
SOR BST EQU N10:0 N9:2 MOV N13:27 C5:4.PRE NXB EQU N10:0 N9:7 MOV N21:21 C5:4.PRE BND EOR
%   N10:0  SYSTEM_STATE  "STATE The current state of the system" %
%   N9:2  SYSTEM_PROCESS  "STATE System Process" %
%   N13:27  REGEN_RUN_TIME %
%   C5:4  REGEN_RUN_MINUTE %
%   N9:7  SYSTEM_COLD_START %
%   N21:21  START_REG_RUN_TIME %
% Rung: 18 %
SOR EQU N13:0 N9:34 BST XIO T4:4/DN TON T4:4 1.0 60 0 NXB XIC T4:4/DN CTU C5:4 480 0 BND EOR
%   N13:0  REGEN_STATE  "STATE The current state of the regen process" %
%   N9:34  REGEN_RUN  "STATE Regen Running" %
%   T4:4  REGEN_RUN_SEC_TMR  "TIMER Regen Run (seconds)" %
%   C5:4  REGEN_RUN_MINUTE %
% Rung: 19 %
SOR EQU N13:0 N9:34 XIC C5:4/DN XIO B34:0/8 MOV N9:35 N13:0 EOR
%   N13:0  REGEN_STATE  "STATE The current state of the regen process" %
%   N9:34  REGEN_RUN  "STATE Regen Running" %
%   C5:4  REGEN_RUN_MINUTE %
%   B34:0/8  SET_REGEN_HOLD %
%   N9:35  REGEN_COOL_WALL  "STATE Regen Cool wall" %

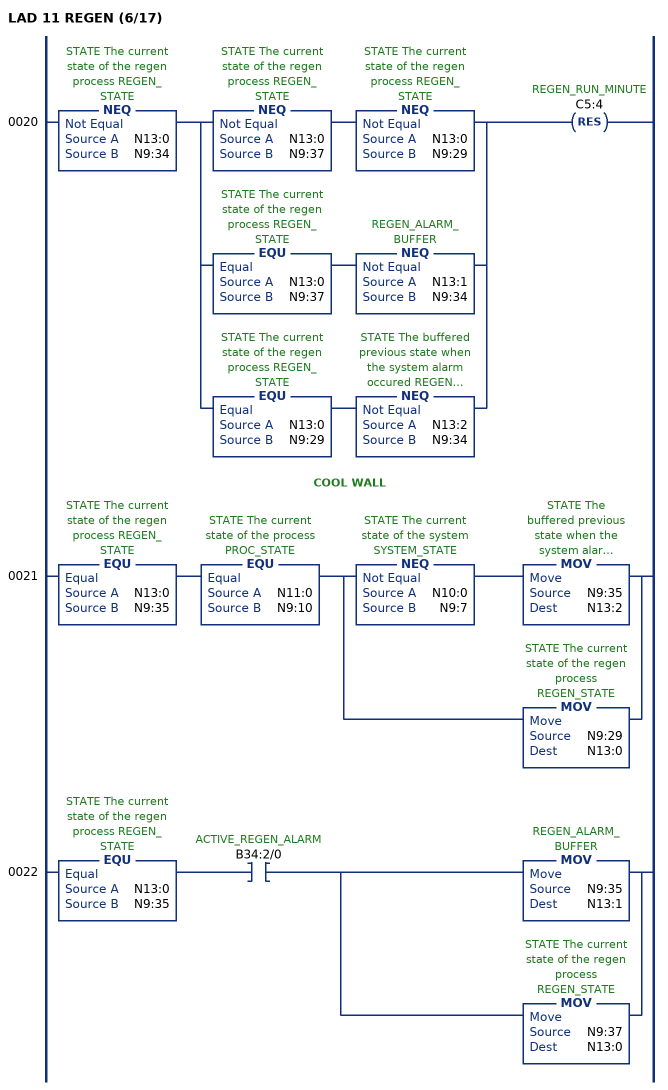
% Rung: 20 %
SOR NEQ N13:0 N9:34 BST NEQ N13:0 N9:37 NEQ N13:0 N9:29 NXB EQU N13:0 N9:37 NEQ N13:1 N9:34 NXB EQU N13:0 N9:29 NEQ N13:2 N9:34 BND RES C5:4 EOR
%   N13:0  REGEN_STATE  "STATE The current state of the regen process" %
%   N9:34  REGEN_RUN  "STATE Regen Running" %
%   N9:37  REGEN_ALARM  "STATE Regen Alarm" %
%   N9:29  REGEN_IDLE %
%   N13:1  REGEN_ALARM_BUFFER %
%   N13:2  REGEN_SYSTEM_BUFFER  "STATE The buffered previous state when the system alarm occured" %
%   C5:4  REGEN_RUN_MINUTE %
% Rung: 21 %
% TITLE: COOL WALL %
SOR EQU N13:0 N9:35 EQU N11:0 N9:10 BST NEQ N10:0 N9:7 MOV N9:35 N13:2 NXB MOV N9:29 N13:0 BND EOR
%   N13:0  REGEN_STATE  "STATE The current state of the regen process" %
%   N9:35  REGEN_COOL_WALL  "STATE Regen Cool wall" %
%   N11:0  PROC_STATE  "STATE The current state of the process" %
%   N9:10  PROC_STANDBY  "STATE Process Standby" %
%   N10:0  SYSTEM_STATE  "STATE The current state of the system" %
%   N9:7  SYSTEM_COLD_START %
%   N13:2  REGEN_SYSTEM_BUFFER  "STATE The buffered previous state when the system alarm occured" %
%   N9:29  REGEN_IDLE %
% Rung: 22 %
SOR EQU N13:0 N9:35 XIC B34:2/0 BST MOV N9:35 N13:1 NXB MOV N9:37 N13:0 BND EOR
%   N13:0  REGEN_STATE  "STATE The current state of the regen process" %
%   N9:35  REGEN_COOL_WALL  "STATE Regen Cool wall" %
%   B34:2/0  ACTIVE_REGEN_ALARM %
%   N13:1  REGEN_ALARM_BUFFER %
%   N9:37  REGEN_ALARM  "STATE Regen Alarm" %

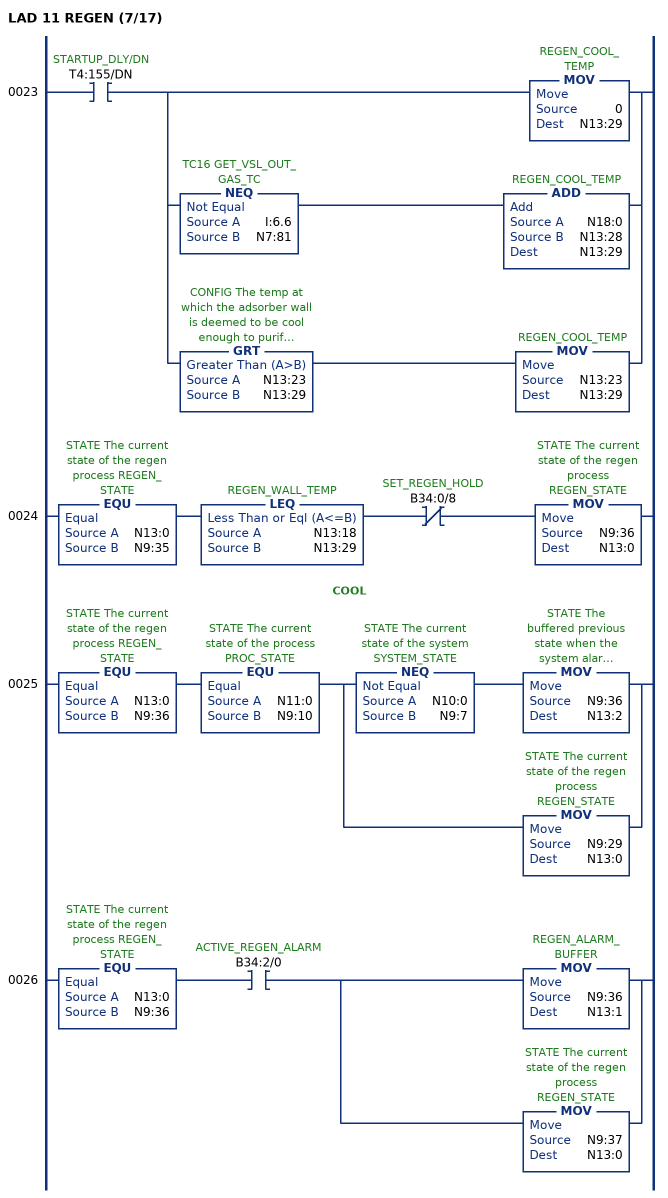
% Rung: 23 %
SOR XIC T4:155/DN BST MOV 0 N13:29 NXB NEQ I:6.6 N7:81 ADD N18:0 N13:28 N13:29 NXB GRT N13:23 N13:29 MOV N13:23 N13:29 BND EOR
%   T4:155  STARTUP_DLY %
%   N13:29  REGEN_COOL_TEMP %
%   I:6.6  GET_VSL_OUT_GAS_TC  "TC16" %
%   N7:81  TC_OPEN_SP  "CONFIG The value read by an open TC input" %
%   N18:0  GET_VSL_OUT_GAS_TEMP %
%   N13:28  REGEN_COOL_DIFF %
%   N13:23  ADS_WALL_TEMP_COOL  "CONFIG The temp at which the adsorber wall is deemed to be cool enough to purify" %
% Rung: 24 %
SOR EQU N13:0 N9:35 LEQ N13:18 N13:29 XIO B34:0/8 MOV N9:36 N13:0 EOR
%   N13:0  REGEN_STATE  "STATE The current state of the regen process" %
%   N9:35  REGEN_COOL_WALL  "STATE Regen Cool wall" %
%   N13:18  REGEN_WALL_TEMP %
%   N13:29  REGEN_COOL_TEMP %
%   B34:0/8  SET_REGEN_HOLD %
%   N9:36  REGEN_COOL  "STATE Regen Cool" %
% Rung: 25 %
% TITLE: COOL %
SOR EQU N13:0 N9:36 EQU N11:0 N9:10 BST NEQ N10:0 N9:7 MOV N9:36 N13:2 NXB MOV N9:29 N13:0 BND EOR
%   N13:0  REGEN_STATE  "STATE The current state of the regen process" %
%   N9:36  REGEN_COOL  "STATE Regen Cool" %
%   N11:0  PROC_STATE  "STATE The current state of the process" %
%   N9:10  PROC_STANDBY  "STATE Process Standby" %
%   N10:0  SYSTEM_STATE  "STATE The current state of the system" %
%   N9:7  SYSTEM_COLD_START %
%   N13:2  REGEN_SYSTEM_BUFFER  "STATE The buffered previous state when the system alarm occured" %
%   N9:29  REGEN_IDLE %
% Rung: 26 %
SOR EQU N13:0 N9:36 XIC B34:2/0 BST MOV N9:36 N13:1 NXB MOV N9:37 N13:0 BND EOR
%   N13:0  REGEN_STATE  "STATE The current state of the regen process" %
%   N9:36  REGEN_COOL  "STATE Regen Cool" %
%   B34:2/0  ACTIVE_REGEN_ALARM %
%   N13:1  REGEN_ALARM_BUFFER %
%   N9:37  REGEN_ALARM  "STATE Regen Alarm" %

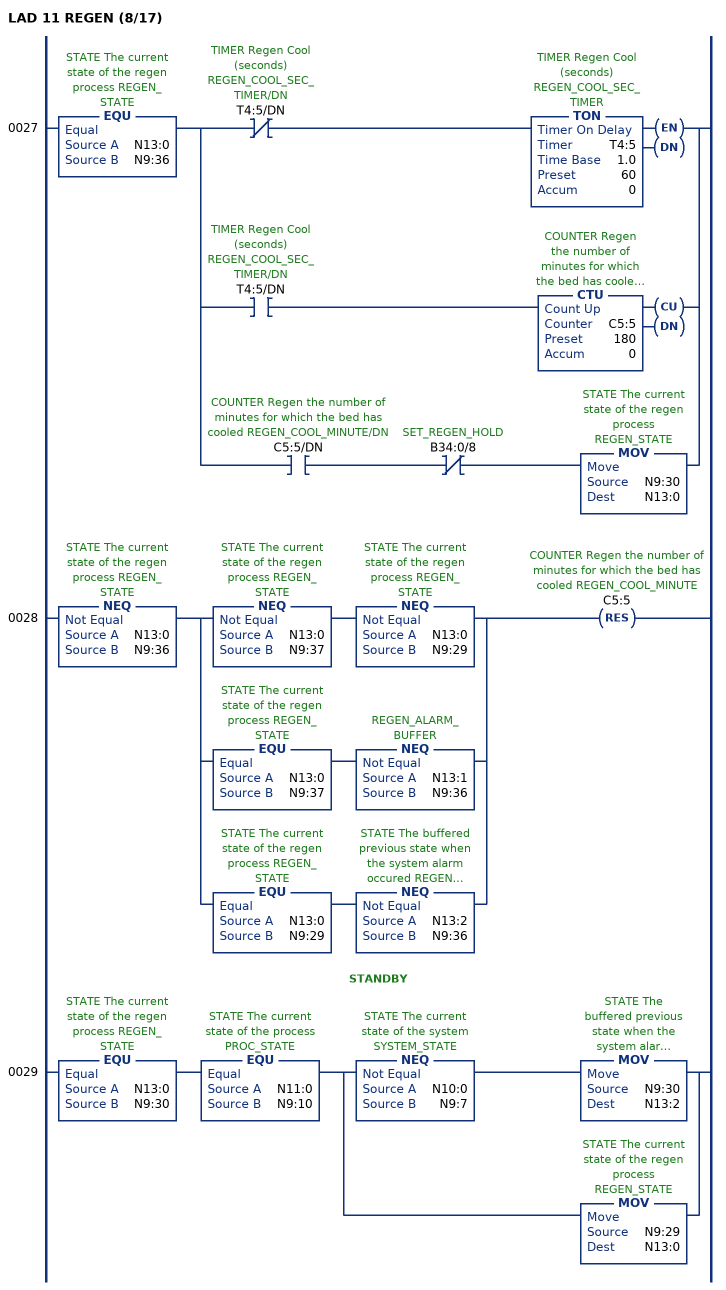
% Rung: 27 %
SOR EQU N13:0 N9:36 BST XIO T4:5/DN TON T4:5 1.0 60 0 NXB XIC T4:5/DN CTU C5:5 180 0 NXB XIC C5:5/DN XIO B34:0/8 MOV N9:30 N13:0 BND EOR
%   N13:0  REGEN_STATE  "STATE The current state of the regen process" %
%   N9:36  REGEN_COOL  "STATE Regen Cool" %
%   T4:5  REGEN_COOL_SEC_TIMER  "TIMER Regen Cool (seconds)" %
%   C5:5  REGEN_COOL_MINUTE  "COUNTER Regen the number of minutes for which the bed has cooled" %
%   B34:0/8  SET_REGEN_HOLD %
%   N9:30  REGEN_STANDBY  "STATE Regen Standby" %
% Rung: 28 %
SOR NEQ N13:0 N9:36 BST NEQ N13:0 N9:37 NEQ N13:0 N9:29 NXB EQU N13:0 N9:37 NEQ N13:1 N9:36 NXB EQU N13:0 N9:29 NEQ N13:2 N9:36 BND RES C5:5 EOR
%   N13:0  REGEN_STATE  "STATE The current state of the regen process" %
%   N9:36  REGEN_COOL  "STATE Regen Cool" %
%   N9:37  REGEN_ALARM  "STATE Regen Alarm" %
%   N9:29  REGEN_IDLE %
%   N13:1  REGEN_ALARM_BUFFER %
%   N13:2  REGEN_SYSTEM_BUFFER  "STATE The buffered previous state when the system alarm occured" %
%   C5:5  REGEN_COOL_MINUTE  "COUNTER Regen the number of minutes for which the bed has cooled" %
% Rung: 29 %
% TITLE: STANDBY %
SOR EQU N13:0 N9:30 EQU N11:0 N9:10 BST NEQ N10:0 N9:7 MOV N9:30 N13:2 NXB MOV N9:29 N13:0 BND EOR
%   N13:0  REGEN_STATE  "STATE The current state of the regen process" %
%   N9:30  REGEN_STANDBY  "STATE Regen Standby" %
%   N11:0  PROC_STATE  "STATE The current state of the process" %
%   N9:10  PROC_STANDBY  "STATE Process Standby" %
%   N10:0  SYSTEM_STATE  "STATE The current state of the system" %
%   N9:7  SYSTEM_COLD_START %
%   N13:2  REGEN_SYSTEM_BUFFER  "STATE The buffered previous state when the system alarm occured" %
%   N9:29  REGEN_IDLE %

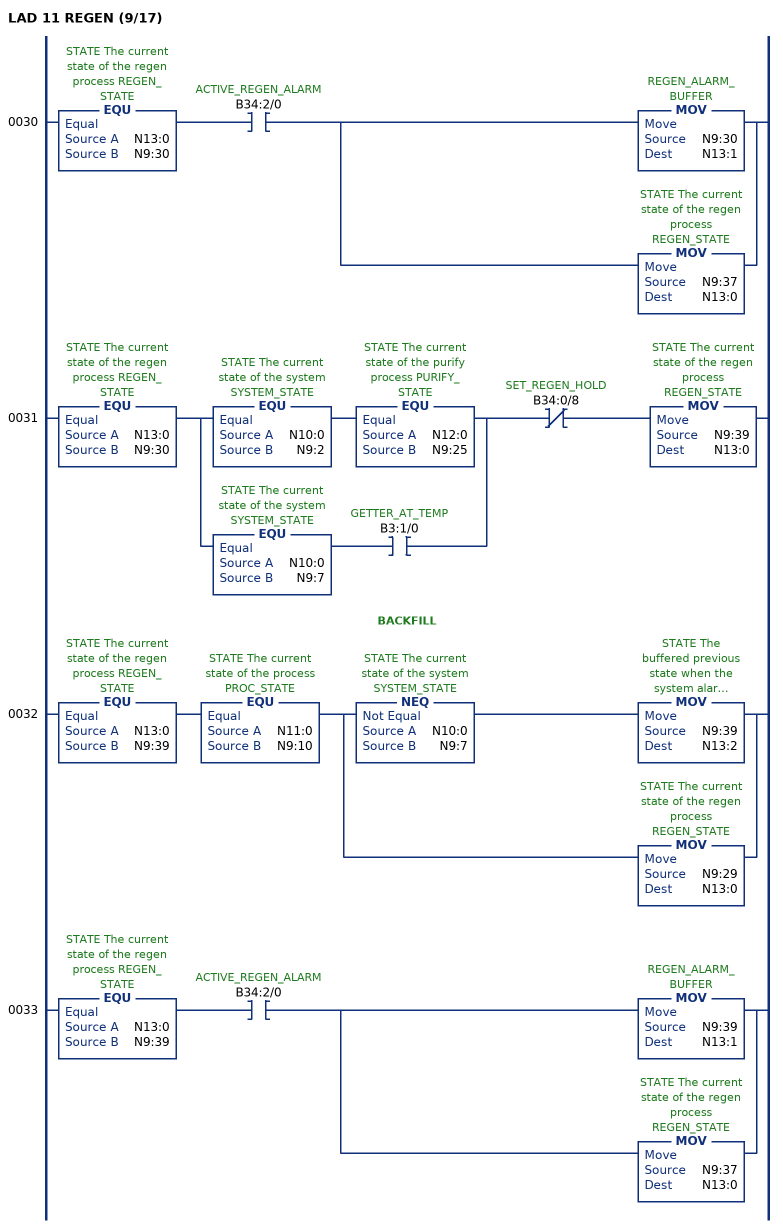
% Rung: 30 %
SOR EQU N13:0 N9:30 XIC B34:2/0 BST MOV N9:30 N13:1 NXB MOV N9:37 N13:0 BND EOR
%   N13:0  REGEN_STATE  "STATE The current state of the regen process" %
%   N9:30  REGEN_STANDBY  "STATE Regen Standby" %
%   B34:2/0  ACTIVE_REGEN_ALARM %
%   N13:1  REGEN_ALARM_BUFFER %
%   N9:37  REGEN_ALARM  "STATE Regen Alarm" %
% Rung: 31 %
SOR EQU N13:0 N9:30 BST EQU N10:0 N9:2 EQU N12:0 N9:25 NXB EQU N10:0 N9:7 XIC B3:1/0 BND XIO B34:0/8 MOV N9:39 N13:0 EOR
%   N13:0  REGEN_STATE  "STATE The current state of the regen process" %
%   N9:30  REGEN_STANDBY  "STATE Regen Standby" %
%   N10:0  SYSTEM_STATE  "STATE The current state of the system" %
%   N9:2  SYSTEM_PROCESS  "STATE System Process" %
%   N12:0  PURIFY_STATE  "STATE The current state of the purify process" %
%   N9:25  PURIFY_DONE %
%   N9:7  SYSTEM_COLD_START %
%   B3:1/0  GETTER_AT_TEMP %
%   B34:0/8  SET_REGEN_HOLD %
%   N9:39  REGEN_BACKFILL %
% Rung: 32 %
% TITLE: BACKFILL %
SOR EQU N13:0 N9:39 EQU N11:0 N9:10 BST NEQ N10:0 N9:7 MOV N9:39 N13:2 NXB MOV N9:29 N13:0 BND EOR
%   N13:0  REGEN_STATE  "STATE The current state of the regen process" %
%   N9:39  REGEN_BACKFILL %
%   N11:0  PROC_STATE  "STATE The current state of the process" %
%   N9:10  PROC_STANDBY  "STATE Process Standby" %
%   N10:0  SYSTEM_STATE  "STATE The current state of the system" %
%   N9:7  SYSTEM_COLD_START %
%   N13:2  REGEN_SYSTEM_BUFFER  "STATE The buffered previous state when the system alarm occured" %
%   N9:29  REGEN_IDLE %
% Rung: 33 %
SOR EQU N13:0 N9:39 XIC B34:2/0 BST MOV N9:39 N13:1 NXB MOV N9:37 N13:0 BND EOR
%   N13:0  REGEN_STATE  "STATE The current state of the regen process" %
%   N9:39  REGEN_BACKFILL %
%   B34:2/0  ACTIVE_REGEN_ALARM %
%   N13:1  REGEN_ALARM_BUFFER %
%   N9:37  REGEN_ALARM  "STATE Regen Alarm" %

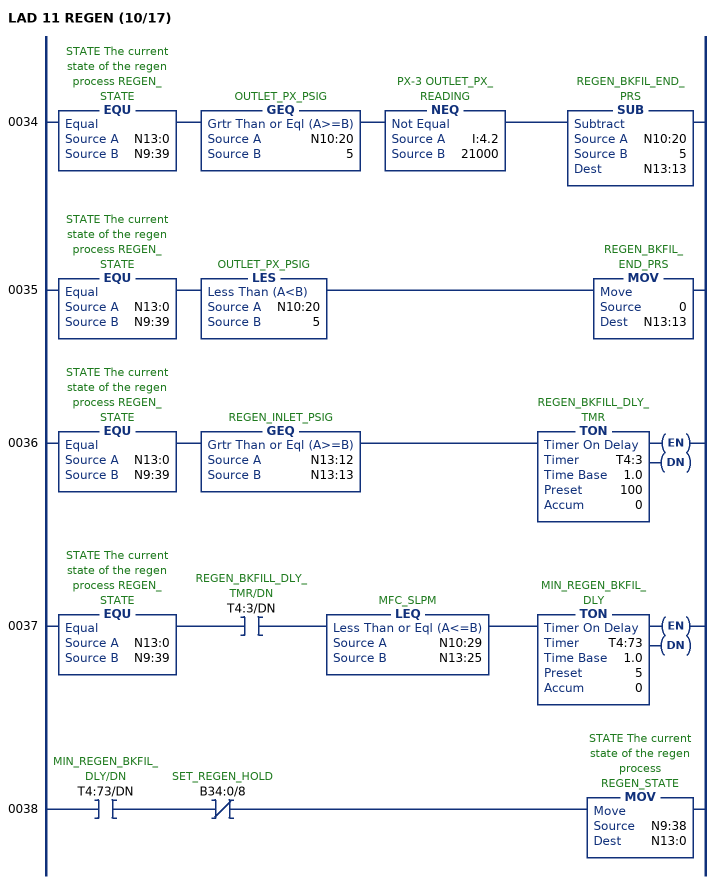
% Rung: 34 %
SOR EQU N13:0 N9:39 GEQ N10:20 5 NEQ I:4.2 21000 SUB N10:20 5 N13:13 EOR
%   N13:0  REGEN_STATE  "STATE The current state of the regen process" %
%   N9:39  REGEN_BACKFILL %
%   N10:20  OUTLET_PX_PSIG %
%   I:4.2  OUTLET_PX_READING  "PX-3" %
%   N13:13  REGEN_BKFIL_END_PRS %
% Rung: 35 %
SOR EQU N13:0 N9:39 LES N10:20 5 MOV 0 N13:13 EOR
%   N13:0  REGEN_STATE  "STATE The current state of the regen process" %
%   N9:39  REGEN_BACKFILL %
%   N10:20  OUTLET_PX_PSIG %
%   N13:13  REGEN_BKFIL_END_PRS %
% Rung: 36 %
SOR EQU N13:0 N9:39 GEQ N13:12 N13:13 TON T4:3 1.0 100 0 EOR
%   N13:0  REGEN_STATE  "STATE The current state of the regen process" %
%   N9:39  REGEN_BACKFILL %
%   N13:12  REGEN_INLET_PSIG %
%   N13:13  REGEN_BKFIL_END_PRS %
%   T4:3  REGEN_BKFILL_DLY_TMR %
% Rung: 37 %
SOR EQU N13:0 N9:39 XIC T4:3/DN LEQ N10:29 N13:25 TON T4:73 1.0 5 0 EOR
%   N13:0  REGEN_STATE  "STATE The current state of the regen process" %
%   N9:39  REGEN_BACKFILL %
%   T4:3  REGEN_BKFILL_DLY_TMR %
%   N10:29  MFC_SLPM %
%   N13:25  REGEN_BKFIL_END_FLOW %
%   T4:73  MIN_REGEN_BKFIL_DLY %
% Rung: 38 %
SOR XIC T4:73/DN XIO B34:0/8 MOV N9:38 N13:0 EOR
%   T4:73  MIN_REGEN_BKFIL_DLY %
%   B34:0/8  SET_REGEN_HOLD %
%   N9:38  REGEN_DONE %
%   N13:0  REGEN_STATE  "STATE The current state of the regen process" %

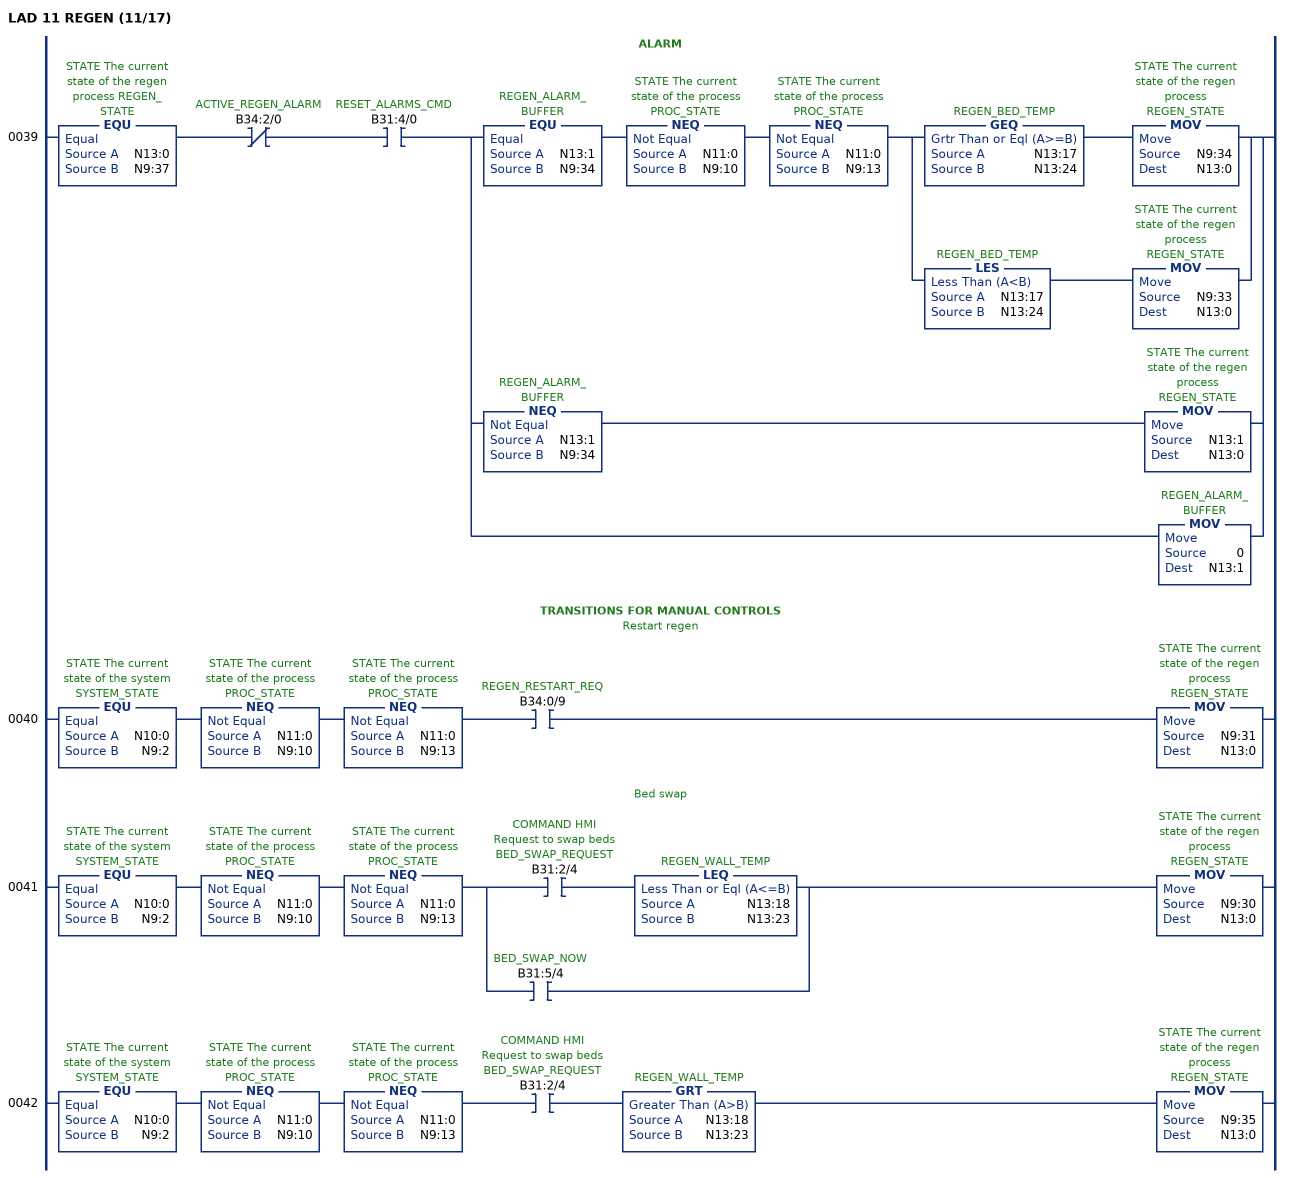
% Rung: 39 %
% TITLE: ALARM %
SOR EQU N13:0 N9:37 XIO B34:2/0 XIC B31:4/0 BST EQU N13:1 N9:34 NEQ N11:0 N9:10 NEQ N11:0 N9:13 BST GEQ N13:17 N13:24 MOV N9:34 N13:0 NXB LES N13:17 N13:24 MOV N9:33 N13:0 BND NXB NEQ N13:1 N9:34 MOV N13:1 N13:0 NXB MOV 0 N13:1 BND EOR
%   N13:0  REGEN_STATE  "STATE The current state of the regen process" %
%   N9:37  REGEN_ALARM  "STATE Regen Alarm" %
%   B34:2/0  ACTIVE_REGEN_ALARM %
%   B31:4/0  RESET_ALARMS_CMD %
%   N13:1  REGEN_ALARM_BUFFER %
%   N9:34  REGEN_RUN  "STATE Regen Running" %
%   N11:0  PROC_STATE  "STATE The current state of the process" %
%   N9:10  PROC_STANDBY  "STATE Process Standby" %
%   N9:13  PROC_OVERLAP  "STATE Process Purify Overlap" %
%   N13:17  REGEN_BED_TEMP %
%   N13:24  ADS_BED_TEMP_HIGH  "CONFIG The temp at which the regen process may continue" %
%   N9:33  REGEN_HEAT_BED  "STATE Regen Heat wall" %
% Rung: 40 %
% TITLE: TRANSITIONS FOR MANUAL CONTROLS %
% Restart regen %
SOR EQU N10:0 N9:2 NEQ N11:0 N9:10 NEQ N11:0 N9:13 XIC B34:0/9 MOV N9:31 N13:0 EOR
%   N10:0  SYSTEM_STATE  "STATE The current state of the system" %
%   N9:2  SYSTEM_PROCESS  "STATE System Process" %
%   N11:0  PROC_STATE  "STATE The current state of the process" %
%   N9:10  PROC_STANDBY  "STATE Process Standby" %
%   N9:13  PROC_OVERLAP  "STATE Process Purify Overlap" %
%   B34:0/9  REGEN_RESTART_REQ %
%   N9:31  REGEN_DELAY  "STATE Regen Delay" %
%   N13:0  REGEN_STATE  "STATE The current state of the regen process" %
% Rung: 41 %
% Bed swap %
SOR EQU N10:0 N9:2 NEQ N11:0 N9:10 NEQ N11:0 N9:13 BST XIC B31:2/4 LEQ N13:18 N13:23 NXB XIC B31:5/4 BND MOV N9:30 N13:0 EOR
%   N10:0  SYSTEM_STATE  "STATE The current state of the system" %
%   N9:2  SYSTEM_PROCESS  "STATE System Process" %
%   N11:0  PROC_STATE  "STATE The current state of the process" %
%   N9:10  PROC_STANDBY  "STATE Process Standby" %
%   N9:13  PROC_OVERLAP  "STATE Process Purify Overlap" %
%   B31:2/4  BED_SWAP_REQUEST  "COMMAND HMI Request to swap beds" %
%   N13:18  REGEN_WALL_TEMP %
%   N13:23  ADS_WALL_TEMP_COOL  "CONFIG The temp at which the adsorber wall is deemed to be cool enough to purify" %
%   B31:5/4  BED_SWAP_NOW %
%   N9:30  REGEN_STANDBY  "STATE Regen Standby" %
%   N13:0  REGEN_STATE  "STATE The current state of the regen process" %
% Rung: 42 %
SOR EQU N10:0 N9:2 NEQ N11:0 N9:10 NEQ N11:0 N9:13 XIC B31:2/4 GRT N13:18 N13:23 MOV N9:35 N13:0 EOR
%   N10:0  SYSTEM_STATE  "STATE The current state of the system" %
%   N9:2  SYSTEM_PROCESS  "STATE System Process" %
%   N11:0  PROC_STATE  "STATE The current state of the process" %
%   N9:10  PROC_STANDBY  "STATE Process Standby" %
%   N9:13  PROC_OVERLAP  "STATE Process Purify Overlap" %
%   B31:2/4  BED_SWAP_REQUEST  "COMMAND HMI Request to swap beds" %
%   N13:18  REGEN_WALL_TEMP %
%   N13:23  ADS_WALL_TEMP_COOL  "CONFIG The temp at which the adsorber wall is deemed to be cool enough to purify" %
%   N9:35  REGEN_COOL_WALL  "STATE Regen Cool wall" %
%   N13:0  REGEN_STATE  "STATE The current state of the regen process" %

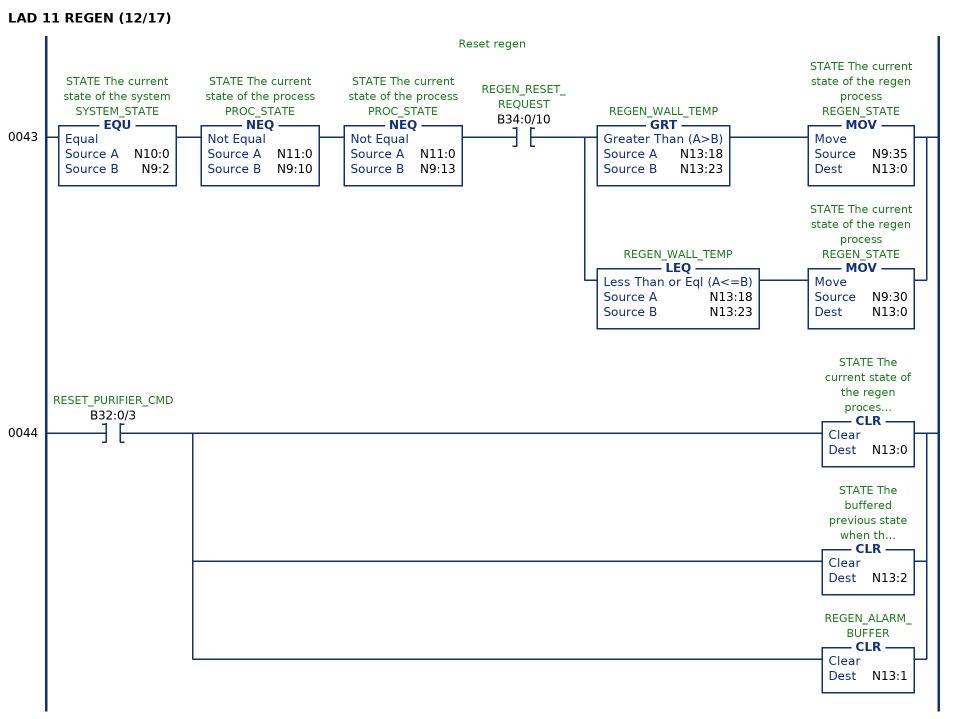
% Rung: 43 %
% Reset regen %
SOR EQU N10:0 N9:2 NEQ N11:0 N9:10 NEQ N11:0 N9:13 XIC B34:0/10 BST GRT N13:18 N13:23 MOV N9:35 N13:0 NXB LEQ N13:18 N13:23 MOV N9:30 N13:0 BND EOR
%   N10:0  SYSTEM_STATE  "STATE The current state of the system" %
%   N9:2  SYSTEM_PROCESS  "STATE System Process" %
%   N11:0  PROC_STATE  "STATE The current state of the process" %
%   N9:10  PROC_STANDBY  "STATE Process Standby" %
%   N9:13  PROC_OVERLAP  "STATE Process Purify Overlap" %
%   B34:0/10  REGEN_RESET_REQUEST %
%   N13:18  REGEN_WALL_TEMP %
%   N13:23  ADS_WALL_TEMP_COOL  "CONFIG The temp at which the adsorber wall is deemed to be cool enough to purify" %
%   N9:35  REGEN_COOL_WALL  "STATE Regen Cool wall" %
%   N13:0  REGEN_STATE  "STATE The current state of the regen process" %
%   N9:30  REGEN_STANDBY  "STATE Regen Standby" %
% Rung: 44 %
SOR XIC B32:0/3 BST CLR N13:0 NXB CLR N13:2 NXB CLR N13:1 BND EOR
%   B32:0/3  RESET_PURIFIER_CMD %
%   N13:0  REGEN_STATE  "STATE The current state of the regen process" %
%   N13:2  REGEN_SYSTEM_BUFFER  "STATE The buffered previous state when the system alarm occured" %
%   N13:1  REGEN_ALARM_BUFFER %

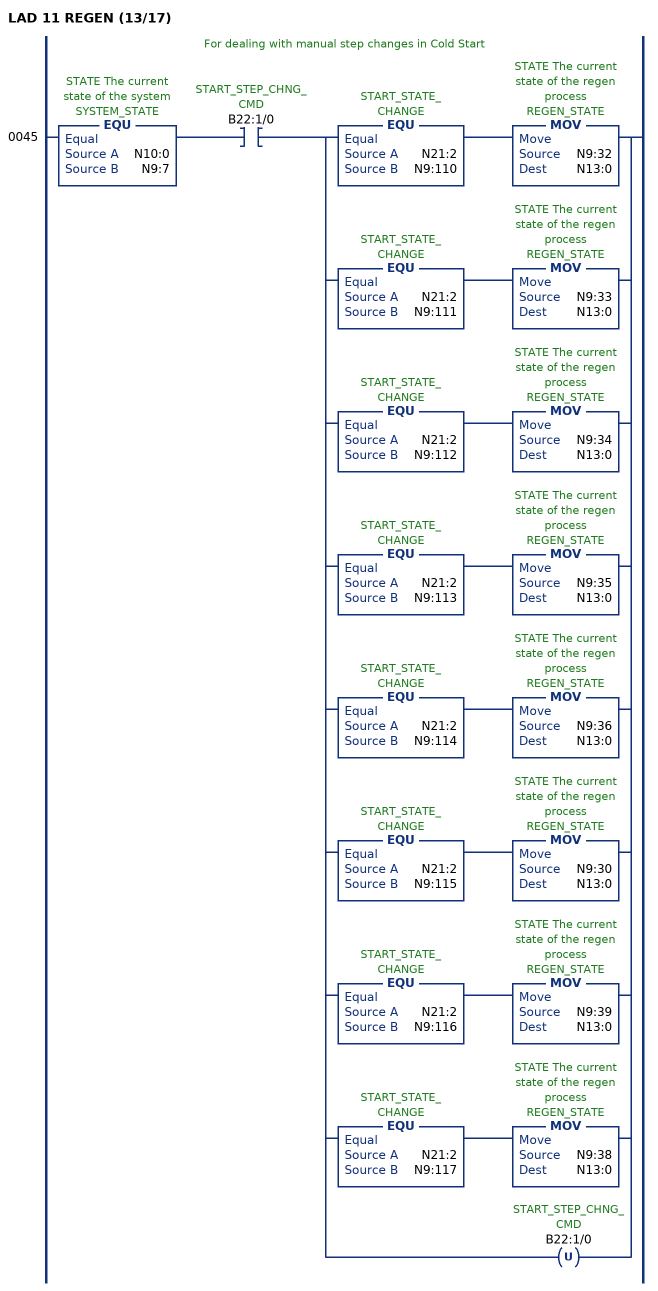
% Rung: 45 %
% For dealing with manual step changes in Cold Start %
SOR EQU N10:0 N9:7 XIC B22:1/0 BST EQU N21:2 N9:110 MOV N9:32 N13:0 NXB EQU N21:2 N9:111 MOV N9:33 N13:0 NXB EQU N21:2 N9:112 MOV N9:34 N13:0 NXB EQU N21:2 N9:113 MOV N9:35 N13:0 NXB EQU N21:2 N9:114 MOV N9:36 N13:0 NXB EQU N21:2 N9:115 MOV N9:30 N13:0 NXB EQU N21:2 N9:116 MOV N9:39 N13:0 NXB EQU N21:2 N9:117 MOV N9:38 N13:0 NXB OTU B22:1/0 BND EOR
%   N10:0  SYSTEM_STATE  "STATE The current state of the system" %
%   N9:7  SYSTEM_COLD_START %
%   B22:1/0  START_STEP_CHNG_CMD %
%   N21:2  START_STATE_CHANGE %
%   N9:110  START_REG_VENT %
%   N9:32  REGEN_VENT  "STATE Regen Vent" %
%   N13:0  REGEN_STATE  "STATE The current state of the regen process" %
%   N9:111  START_REG_HEAT %
%   N9:33  REGEN_HEAT_BED  "STATE Regen Heat wall" %
%   N9:112  START_REG_RUN %
%   N9:34  REGEN_RUN  "STATE Regen Running" %
%   N9:113  START_REG_COOL %
%   N9:35  REGEN_COOL_WALL  "STATE Regen Cool wall" %
%   N9:114  START_REG_TIMED_COOL %
%   N9:36  REGEN_COOL  "STATE Regen Cool" %
%   N9:115  START_REG_STANDBY %
%   N9:30  REGEN_STANDBY  "STATE Regen Standby" %
%   N9:116  START_REG_BACKFILL %
%   N9:39  REGEN_BACKFILL %
%   N9:117  START_REG_DONE %
%   N9:38  REGEN_DONE %

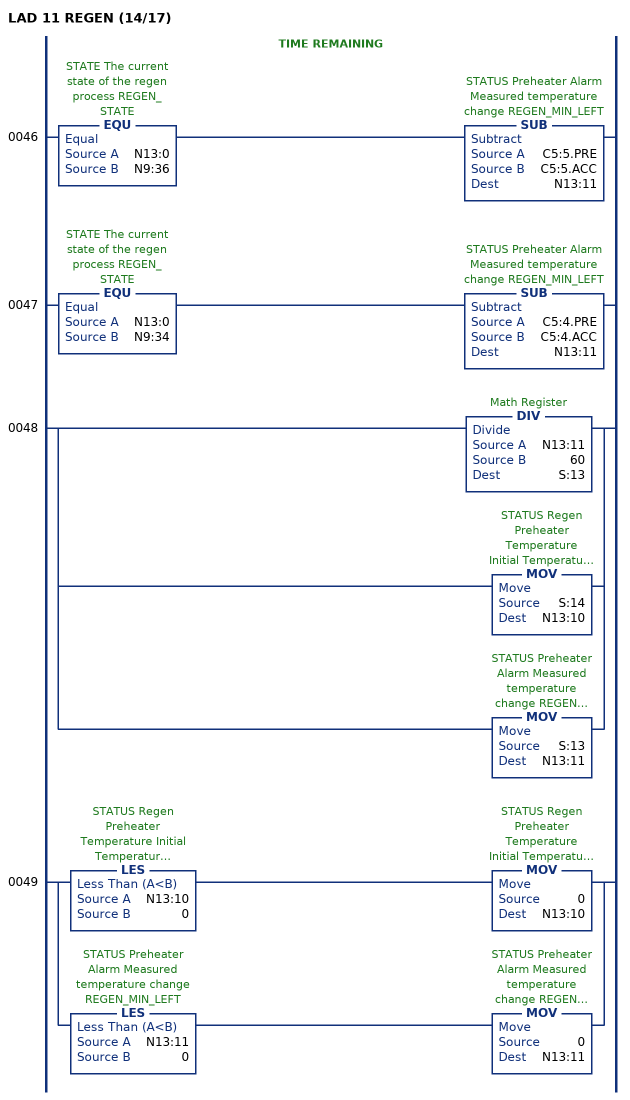
% Rung: 46 %
% TITLE: TIME REMAINING %
SOR EQU N13:0 N9:36 SUB C5:5.PRE C5:5.ACC N13:11 EOR
%   N13:0  REGEN_STATE  "STATE The current state of the regen process" %
%   N9:36  REGEN_COOL  "STATE Regen Cool" %
%   C5:5  REGEN_COOL_MINUTE  "COUNTER Regen the number of minutes for which the bed has cooled" %
%   N13:11  REGEN_MIN_LEFT  "STATUS Preheater Alarm Measured temperature change" %
% Rung: 47 %
SOR EQU N13:0 N9:34 SUB C5:4.PRE C5:4.ACC N13:11 EOR
%   N13:0  REGEN_STATE  "STATE The current state of the regen process" %
%   N9:34  REGEN_RUN  "STATE Regen Running" %
%   C5:4  REGEN_RUN_MINUTE %
%   N13:11  REGEN_MIN_LEFT  "STATUS Preheater Alarm Measured temperature change" %
% Rung: 48 %
SOR BST DIV N13:11 60 S:13 NXB MOV S:14 N13:10 NXB MOV S:13 N13:11 BND EOR
%   N13:11  REGEN_MIN_LEFT  "STATUS Preheater Alarm Measured temperature change" %
%   S:13  "Math Register" %
%   S:14  "Math Register" %
%   N13:10  REGEN_HRS_LEFT  "STATUS Regen Preheater Temperature Initial Temperature" %
% Rung: 49 %
SOR BST LES N13:10 0 MOV 0 N13:10 NXB LES N13:11 0 MOV 0 N13:11 BND EOR
%   N13:10  REGEN_HRS_LEFT  "STATUS Regen Preheater Temperature Initial Temperature" %
%   N13:11  REGEN_MIN_LEFT  "STATUS Preheater Alarm Measured temperature change" %

